KUKA KRL program: EPS_2_25716_MHDR03_A_20250926070354.src

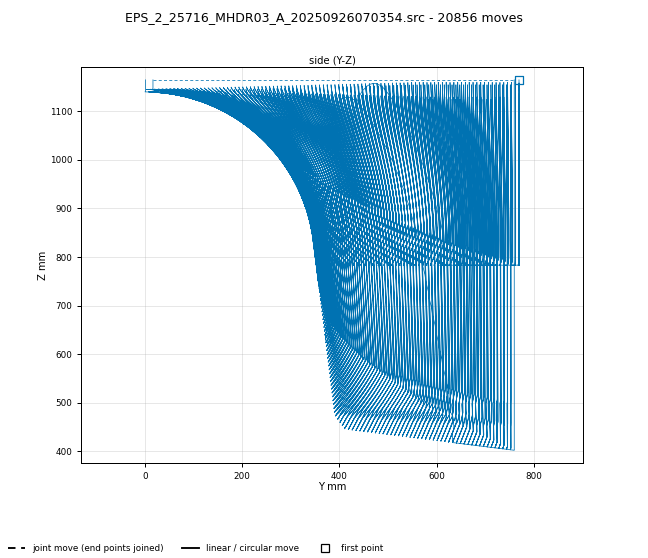
[picture p0: tool path of EPS_2_25716_MHDR03_A_20250926070354.src, 20856 of 20858 moves have a stored position in this frame; points joined in program order, loops and branches not executed]
&ACCESS RVP
&REL 4
&COMMENT QRS 19112012
&PARAM EDITMASK = *
DEF PART()
EXT BAS (BAS_COMMAND :IN,REAL :IN )
INT I
BAS (#INITMOV,0 )

;KUKA QRS Post kuka4.cps  Date:22-06-2017 !

File_ID=2852

QRS_PRE_INIT()

;Init var - Until changes are made in qrs_pre_init
Outlet_Square_prg=0
Inlet_1_Square_prg=0
Inlet_2_Square_prg=0
Inlet_3_Square_prg=0
Inlet_4_Square_prg=0
Inlet_5_Square_prg=0

Outlet_1={X 0.000, Y 562.000, Z 811.500, B 0.000, E1 0.000 }
Inlet_1={X 0.000, Y 582.000, Z 819.500, B 0.000, E1 180.000 }
Outlet_1_type=686
Inlet_1_type=610
;QRS#1=Sidecore dimensions
;QRS#2=675-27" Concrete
;QRS#3=600-24" Concrete
;QRS#4=
;QRS#5=
;QRS#6=
;QRS#7=
;QRS#8=
;QRS#9=S306-38L
;QRS#10=S306-34L
;QRS#11=
;QRS#12=
;QRS#13=
;QRS#14=
;QRS#15=
;QRS#16=1524x152x1600 5,25'
;QRS#17=EPS Height
;QRS#18=1154,5
;QRS#19=*
;QRS#20= UPDATED VERSION 22-06-2017
;QRS#21=*
Outlet_Square=0550
Inlet_1_Square=0450
Inlet_2_Square=0
Inlet_3_Square=0
Inlet_4_Square=0
Inlet_5_Square=0
Mill_Square=1
Outlet_Square_Prg=265
Inlet_1_Square_prg=264

QRS_INIT()

$ADVANCE=5

; T1
PTP {E1 171.915,E2 171.915}
PTP {X 0,Y 769.686,A -85,B 0,C 180,E1 171.915,E2 171.915,E3 0,E4 0,E5 0,E6 0}
QRS_SPEED_INIT()
LIN {X 0,Y 769.686,Z 1164.5,A -85,B 0,C 180,E1 171.915,E2 171.915,E3 0,E4 0,E5 0,E6 0} C_VEL
LIN {X 0,Y 769.686,Z 785.31,A -85,B 0,C 180,E1 171.915,E2 171.915} C_VEL
LIN {X 0,Y 769.694,Z 783.31,A -85,B 0,C 180,E1 172.064,E2 172.064} C_VEL
LIN {X 0,Y 770.026,Z 783.31,A -85,B 0,C 180,E1 173.477,E2 173.477} C_VEL
LIN {X 0,Y 770.008,Z 783.31,A -85,B 0,C 180,E1 177.209,E2 177.209} C_VEL
LIN {X 0,Y 770.018,Z 783.31,A -85,B 0,C 180,E1 180.93,E2 180.93} C_VEL
LIN {X 0,Y 769.994,Z 783.31,A -85,B 0,C 180,E1 184.655,E2 184.655} C_VEL
LIN {X 0,Y 770.012,Z 783.31,A -85,B 0,C 180,E1 188.399,E2 188.399} C_VEL
LIN {X 0,Y 770.006,Z 783.31,A -85,B 0,C 180,E1 192.18,E2 192.18} C_VEL
LIN {X 0,Y 769.997,Z 783.31,A -85,B 0,C 180,E1 196.016,E2 196.016} C_VEL
LIN {X 0,Y 769.871,Z 783.31,A -85,B 0,C 180,E1 196.719,E2 196.719} C_VEL
LIN {X 0,Y 769.991,Z 783.31,A -85,B 0,C 180,E1 199.928,E2 199.928} C_VEL
LIN {X 0,Y 769.967,Z 783.31,A -85,B 0,C 180,E1 203.939,E2 203.939} C_VEL
LIN {X 0,Y 769.591,Z 783.31,A -85,B 0,C 180,E1 206.732,E2 206.732} C_VEL
LIN {X 0,Y 769.94,Z 783.31,A -85,B 0,C 180,E1 208.08,E2 208.08} C_VEL
LIN {X 0,Y 769.516,Z 783.31,A -85,B 0,C 180,E1 210.601,E2 210.601} C_VEL
LIN {X 0,Y 769.912,Z 783.31,A -85,B 0,C 180,E1 212.388,E2 212.388} C_VEL
LIN {X 0,Y 769.473,Z 783.31,A -85,B 0,C 180,E1 214.641,E2 214.641} C_VEL
LIN {X 0,Y 770.033,Z 783.31,A -85,B 0,C 180,E1 217.323,E2 217.323} C_VEL
LIN {X 0,Y 769.708,Z 783.31,A -85,B 0,C 180,E1 221.735,E2 221.735} C_VEL
LIN {X 0,Y 769.752,Z 783.31,A -85,B 0,C 180,E1 223.065,E2 223.065} C_VEL
LIN {X 0,Y 769.737,Z 783.31,A -85,B 0,C 180,E1 226.937,E2 226.937} C_VEL
LIN {X 0,Y 769.694,Z 783.31,A -85,B 0,C 180,E1 228.264,E2 228.264} C_VEL
LIN {X 0,Y 770.056,Z 783.31,A -85,B 0,C 180,E1 232.675,E2 232.675} C_VEL
LIN {X 0,Y 769.726,Z 783.31,A -85,B 0,C 180,E1 235.896,E2 235.896} C_VEL
LIN {X 0,Y 769.776,Z 783.31,A -85,B 0,C 180,E1 237.606,E2 237.606} C_VEL
LIN {X 0,Y 770.022,Z 783.31,A -85,B 0,C 180,E1 240.257,E2 240.257} C_VEL
LIN {X 0,Y 769.768,Z 783.31,A -85,B 0,C 180,E1 240.477,E2 240.477} C_VEL
LIN {X 0,Y 767.999,Z 783.31,A -85,B 0,C 180,E1 240.652,E2 240.652} C_VEL
LIN {X 0,Y 768.022,Z 783.933,A -85,B 0,C 180,E1 240.678,E2 240.678} C_VEL
LIN {X 0,Y 769.268,Z 788.284,A -85,B 0,C 180,E1 240.775,E2 240.775} C_VEL
LIN {X 0,Y 769.55,Z 789.73,A -85,B 0,C 180,E1 240.802,E2 240.802} C_VEL
LIN {X 0,Y 769.707,Z 828.612,A -85,B 0,C 180,E1 241.215,E2 241.215} C_VEL
LIN {X 0,Y 769.834,Z 848.893,A -85,B 0,C 180,E1 241.465,E2 241.465} C_VEL
LIN {X 0,Y 769.636,Z 866.973,A -85,B 0,C 180,E1 241.758,E2 241.758} C_VEL
LIN {X 0,Y 769.793,Z 884.542,A -85,B 0,C 180,E1 242.131,E2 242.131} C_VEL
LIN {X 0,Y 769.673,Z 901.057,A -85,B 0,C 180,E1 242.539,E2 242.539} C_VEL
LIN {X 0,Y 769.87,Z 917.184,A -85,B 0,C 180,E1 243.017,E2 243.017} C_VEL
LIN {X 0,Y 769.856,Z 933.115,A -85,B 0,C 180,E1 243.548,E2 243.548} C_VEL
LIN {X 0,Y 769.816,Z 943.907,A -85,B 0,C 180,E1 243.947,E2 243.947} C_VEL
LIN {X 0,Y 769.91,Z 958.612,A -85,B 0,C 180,E1 244.549,E2 244.549} C_VEL
LIN {X 0,Y 769.91,Z 966.436,A -85,B 0,C 180,E1 244.896,E2 244.896} C_VEL
LIN {X 0,Y 769.862,Z 978.838,A -85,B 0,C 180,E1 245.477,E2 245.477} C_VEL
LIN {X 0,Y 769.916,Z 992.577,A -85,B 0,C 180,E1 246.186,E2 246.186} C_VEL
LIN {X 0,Y 769.931,Z 1006.072,A -85,B 0,C 180,E1 246.947,E2 246.947} C_VEL
LIN {X 0,Y 769.916,Z 1018.978,A -85,B 0,C 180,E1 247.739,E2 247.739} C_VEL
LIN {X 0,Y 769.895,Z 1031.838,A -85,B 0,C 180,E1 248.599,E2 248.599} C_VEL
LIN {X 0,Y 769.943,Z 1043.698,A -85,B 0,C 180,E1 249.463,E2 249.463} C_VEL
LIN {X 0,Y 769.918,Z 1056.014,A -85,B 0,C 180,E1 250.441,E2 250.441} C_VEL
LIN {X 0,Y 769.89,Z 1066.051,A -85,B 0,C 180,E1 251.302,E2 251.302} C_VEL
LIN {X 0,Y 769.98,Z 1077.133,A -85,B 0,C 180,E1 252.343,E2 252.343} C_VEL
LIN {X 0,Y 769.834,Z 1086.51,A -85,B 0,C 180,E1 253.29,E2 253.29} C_VEL
LIN {X 0,Y 769.849,Z 1096.259,A -85,B 0,C 180,E1 254.375,E2 254.375} C_VEL
LIN {X 0,Y 769.966,Z 1105.17,A -85,B 0,C 180,E1 255.468,E2 255.468} C_VEL
LIN {X 0,Y 769.773,Z 1113.783,A -85,B 0,C 180,E1 256.624,E2 256.624} C_VEL
LIN {X 0,Y 769.792,Z 1120.236,A -85,B 0,C 180,E1 257.578,E2 257.578} C_VEL
LIN {X 0,Y 769.971,Z 1127.408,A -85,B 0,C 180,E1 258.769,E2 258.769} C_VEL
LIN {X 0,Y 769.802,Z 1133.795,A -85,B 0,C 180,E1 259.949,E2 259.949} C_VEL
LIN {X 0,Y 769.935,Z 1140.321,A -85,B 0,C 180,E1 261.365,E2 261.365} C_VEL
LIN {X 0,Y 769.915,Z 1143.557,A -85,B 0,C 180,E1 262.172,E2 262.172} C_VEL
LIN {X 0,Y 769.781,Z 1146.098,A -85,B 0,C 180,E1 262.858,E2 262.858} C_VEL
LIN {X 0,Y 769.778,Z 1149.359,A -85,B 0,C 180,E1 263.849,E2 263.849} C_VEL
LIN {X 0,Y 769.874,Z 1151.367,A -85,B 0,C 180,E1 264.598,E2 264.598} C_VEL
LIN {X 0,Y 769.914,Z 1153.173,A -85,B 0,C 180,E1 265.345,E2 265.345} C_VEL
LIN {X 0,Y 769.718,Z 1155.452,A -85,B 0,C 180,E1 266.463,E2 266.463} C_VEL
LIN {X 0,Y 769.72,Z 1156.563,A -85,B 0,C 180,E1 267.208,E2 267.208} C_VEL
LIN {X 0,Y 769.828,Z 1157.375,A -85,B 0,C 180,E1 267.953,E2 267.953} C_VEL
LIN {X 0,Y 769.875,Z 1158.173,A -85,B 0,C 180,E1 269.07,E2 269.07} C_VEL
LIN {X 0,Y 769.75,Z 1158.207,A -85,B 0,C 180,E1 270.93,E2 270.93} C_VEL
LIN {X 0,Y 769.983,Z 1157.332,A -85,B 0,C 180,E1 272.046,E2 272.046} C_VEL
LIN {X 0,Y 769.854,Z 1156.527,A -85,B 0,C 180,E1 272.791,E2 272.791} C_VEL
LIN {X 0,Y 769.764,Z 1155.44,A -85,B 0,C 180,E1 273.537,E2 273.537} C_VEL
LIN {X 0,Y 769.915,Z 1152.382,A -85,B 0,C 180,E1 275.029,E2 275.029} C_VEL
LIN {X 0,Y 769.886,Z 1150.344,A -85,B 0,C 180,E1 275.776,E2 275.776} C_VEL
LIN {X 0,Y 769.765,Z 1148.176,A -85,B 0,C 180,E1 276.525,E2 276.525} C_VEL
LIN {X 0,Y 769.743,Z 1145.274,A -85,B 0,C 180,E1 277.392,E2 277.392} C_VEL
LIN {X 0,Y 769.948,Z 1139.305,A -85,B 0,C 180,E1 278.87,E2 278.87} C_VEL
LIN {X 0,Y 769.75,Z 1133.807,A -85,B 0,C 180,E1 280.051,E2 280.051} C_VEL
LIN {X 0,Y 769.818,Z 1127.44,A -85,B 0,C 180,E1 281.233,E2 281.233} C_VEL
LIN {X 0,Y 769.954,Z 1121.667,A -85,B 0,C 180,E1 282.181,E2 282.181} C_VEL
LIN {X 0,Y 769.843,Z 1116.993,A -85,B 0,C 180,E1 282.897,E2 282.897} C_VEL
LIN {X 0,Y 769.807,Z 1112.103,A -85,B 0,C 180,E1 283.615,E2 283.615} C_VEL
LIN {X 0,Y 769.951,Z 1102.998,A -85,B 0,C 180,E1 284.806,E2 284.806} C_VEL
LIN {X 0,Y 769.846,Z 1094.002,A -85,B 0,C 180,E1 285.885,E2 285.885} C_VEL
LIN {X 0,Y 769.836,Z 1084.723,A -85,B 0,C 180,E1 286.898,E2 286.898} C_VEL
LIN {X 0,Y 769.967,Z 1073.994,A -85,B 0,C 180,E1 287.962,E2 287.962} C_VEL
LIN {X 0,Y 769.883,Z 1063.259,A -85,B 0,C 180,E1 288.944,E2 288.944} C_VEL
LIN {X 0,Y 769.915,Z 1053.038,A -85,B 0,C 180,E1 289.806,E2 289.806} C_VEL
LIN {X 0,Y 769.961,Z 1041.658,A -85,B 0,C 180,E1 290.69,E2 290.69} C_VEL
LIN {X 0,Y 769.906,Z 1029.266,A -85,B 0,C 180,E1 291.578,E2 291.578} C_VEL
LIN {X 0,Y 769.903,Z 1016.603,A -85,B 0,C 180,E1 292.412,E2 292.412} C_VEL
LIN {X 0,Y 769.92,Z 1002.799,A -85,B 0,C 180,E1 293.243,E2 293.243} C_VEL
LIN {X 0,Y 769.909,Z 988.614,A -85,B 0,C 180,E1 294.024,E2 294.024} C_VEL
LIN {X 0,Y 769.846,Z 975.459,A -85,B 0,C 180,E1 294.69,E2 294.69} C_VEL
LIN {X 0,Y 769.908,Z 960.966,A -85,B 0,C 180,E1 295.353,E2 295.353} C_VEL
LIN {X 0,Y 769.866,Z 944.041,A -85,B 0,C 180,E1 296.047,E2 296.047} C_VEL
LIN {X 0,Y 769.796,Z 931.365,A -85,B 0,C 180,E1 296.519,E2 296.519} C_VEL
LIN {X 0,Y 769.894,Z 913.334,A -85,B 0,C 180,E1 297.102,E2 297.102} C_VEL
LIN {X 0,Y 769.78,Z 896.592,A -85,B 0,C 180,E1 297.576,E2 297.576} C_VEL
LIN {X 0,Y 769.701,Z 887.337,A -85,B 0,C 180,E1 297.804,E2 297.804} C_VEL
LIN {X 0,Y 769.825,Z 878.224,A -85,B 0,C 180,E1 298.006,E2 298.006} C_VEL
LIN {X 0,Y 769.846,Z 863.646,A -85,B 0,C 180,E1 298.294,E2 298.294} C_VEL
LIN {X 0,Y 769.602,Z 846.73,A -85,B 0,C 180,E1 298.572,E2 298.572} C_VEL
LIN {X 0,Y 769.68,Z 827.338,A -85,B 0,C 180,E1 298.799,E2 298.799} C_VEL
LIN {X 0,Y 769.587,Z 792.326,A -85,B 0,C 180,E1 299.169,E2 299.169} C_VEL
LIN {X 0,Y 769.462,Z 789.243,A -85,B 0,C 180,E1 299.206,E2 299.206} C_VEL
LIN {X 0,Y 768.376,Z 784.955,A -85,B 0,C 180,E1 299.297,E2 299.297} C_VEL
LIN {X 0,Y 767.908,Z 783.31,A -85,B 0,C 180,E1 299.343,E2 299.343} C_VEL
LIN {X 0,Y 769.576,Z 783.31,A -85,B 0,C 180,E1 299.487,E2 299.487} C_VEL
LIN {X 0,Y 770.036,Z 783.31,A -85,B 0,C 180,E1 299.696,E2 299.696} C_VEL
LIN {X 0,Y 769.963,Z 783.31,A -85,B 0,C 180,E1 302.386,E2 302.386} C_VEL
LIN {X 0,Y 769.484,Z 783.31,A -85,B 0,C 180,E1 304.641,E2 304.641} C_VEL
LIN {X 0,Y 770.058,Z 783.31,A -85,B 0,C 180,E1 307.325,E2 307.325} C_VEL
LIN {X 0,Y 769.794,Z 783.31,A -85,B 0,C 180,E1 311.729,E2 311.729} C_VEL
LIN {X 0,Y 769.849,Z 783.31,A -85,B 0,C 180,E1 313.072,E2 313.072} C_VEL
LIN {X 0,Y 769.85,Z 783.31,A -85,B 0,C 180,E1 314.269,E2 314.269} C_VEL
LIN {X 0,Y 769.763,Z 783.31,A -85,B 0,C 180,E1 315.725,E2 315.725} C_VEL
LIN {X 0,Y 769.779,Z 783.31,A -85,B 0,C 180,E1 319.732,E2 319.732} C_VEL
LIN {X 0,Y 769.826,Z 783.31,A -85,B 0,C 180,E1 320.72,E2 320.72} C_VEL
LIN {X 0,Y 769.435,Z 783.31,A -85,B 0,C 180,E1 323.062,E2 323.062} C_VEL
LIN {X 0,Y 769.867,Z 783.31,A -85,B 0,C 180,E1 325.379,E2 325.379} C_VEL
LIN {X 0,Y 770.015,Z 783.31,A -85,B 0,C 180,E1 329.336,E2 329.336} C_VEL
LIN {X 0,Y 769.861,Z 783.31,A -85,B 0,C 180,E1 333.228,E2 333.228} C_VEL
LIN {X 0,Y 769.954,Z 783.31,A -85,B 0,C 180,E1 334.009,E2 334.009} C_VEL
LIN {X 0,Y 770.01,Z 783.31,A -85,B 0,C 180,E1 337.683,E2 337.683} C_VEL
LIN {X 0,Y 769.98,Z 783.31,A -85,B 0,C 180,E1 338.081,E2 338.081} C_VEL
LIN {X 0,Y 770,Z 783.31,A -85,B 0,C 180,E1 342.039,E2 342.039} C_VEL
LIN {X 0,Y 769.707,Z 783.31,A -85,B 0,C 180,E1 343.978,E2 343.978} C_VEL
LIN {X 0,Y 769.796,Z 783.31,A -85,B 0,C 180,E1 345.906,E2 345.906} C_VEL
LIN {X 0,Y 770.015,Z 783.31,A -85,B 0,C 180,E1 349.716,E2 349.716} C_VEL
LIN {X 0,Y 769.998,Z 783.31,A -85,B 0,C 180,E1 353.477,E2 353.477} C_VEL
LIN {X 0,Y 770.007,Z 783.31,A -85,B 0,C 180,E1 357.209,E2 357.209} C_VEL
LIN {X 0,Y 769.992,Z 783.31,A -85,B 0,C 180,E1 360.93,E2 360.93} C_VEL
LIN {X 0,Y 770.022,Z 783.31,A -85,B 0,C 180,E1 364.655,E2 364.655} C_VEL
LIN {X 0,Y 770.009,Z 783.31,A -85,B 0,C 180,E1 368.399,E2 368.399} C_VEL
LIN {X 0,Y 770.002,Z 783.31,A -85,B 0,C 180,E1 372.18,E2 372.18} C_VEL
LIN {X 0,Y 769.963,Z 783.31,A -85,B 0,C 180,E1 376.017,E2 376.017} C_VEL
LIN {X 0,Y 769.575,Z 783.31,A -85,B 0,C 180,E1 377.971,E2 377.971} C_VEL
LIN {X 0,Y 769.931,Z 783.31,A -85,B 0,C 180,E1 379.929,E2 379.929} C_VEL
LIN {X 0,Y 769.547,Z 783.31,A -85,B 0,C 180,E1 382.233,E2 382.233} C_VEL
LIN {X 0,Y 769.894,Z 783.31,A -85,B 0,C 180,E1 383.942,E2 383.942} C_VEL
LIN {X 0,Y 769.539,Z 783.31,A -85,B 0,C 180,E1 386.724,E2 386.724} C_VEL
LIN {X 0,Y 769.895,Z 783.31,A -85,B 0,C 180,E1 388.082,E2 388.082} C_VEL
LIN {X 0,Y 769.51,Z 783.31,A -85,B 0,C 180,E1 390.601,E2 390.601} C_VEL
LIN {X 0,Y 769.898,Z 783.31,A -85,B 0,C 180,E1 392.389,E2 392.389} C_VEL
LIN {X 0,Y 769.447,Z 783.31,A -85,B 0,C 180,E1 394.643,E2 394.643} C_VEL
LIN {X 0,Y 769.995,Z 783.31,A -85,B 0,C 180,E1 397.319,E2 397.319} C_VEL
LIN {X 0,Y 769.732,Z 783.31,A -85,B 0,C 180,E1 401.733,E2 401.733} C_VEL
LIN {X 0,Y 769.804,Z 783.31,A -85,B 0,C 180,E1 403.069,E2 403.069} C_VEL
LIN {X 0,Y 769.812,Z 783.31,A -85,B 0,C 180,E1 404.272,E2 404.272} C_VEL
LIN {X 0,Y 769.735,Z 783.31,A -85,B 0,C 180,E1 405.723,E2 405.723} C_VEL
LIN {X 0,Y 769.736,Z 783.31,A -85,B 0,C 180,E1 409.736,E2 409.736} C_VEL
LIN {X 0,Y 769.771,Z 783.31,A -85,B 0,C 180,E1 410.717,E2 410.717} C_VEL
LIN {X 0,Y 769.411,Z 783.31,A -85,B 0,C 180,E1 413.061,E2 413.061} C_VEL
LIN {X 0,Y 769.871,Z 783.31,A -85,B 0,C 180,E1 415.379,E2 415.379} C_VEL
LIN {X 0,Y 770.03,Z 783.31,A -85,B 0,C 180,E1 419.334,E2 419.334} C_VEL
LIN {X 0,Y 769.98,Z 783.31,A -85,B 0,C 180,E1 423.211,E2 423.211} C_VEL
LIN {X 0,Y 769.96,Z 783.31,A -85,B 0,C 180,E1 423.598,E2 423.598} C_VEL
LIN {X 0,Y 769.249,Z 783.341,A -85,B 0,C 180,E1 423.817,E2 423.817} C_VEL
LIN {X 0,Y 769.67,Z 784.885,A -85,B 0,C 180,E1 423.848,E2 423.848} C_VEL
LIN {X 0,Y 769.75,Z 839.545,A -85,B 0,C 180,E1 424.413,E2 424.413} C_VEL
LIN {X 0,Y 769.691,Z 849.688,A -85,B 0,C 180,E1 424.533,E2 424.533} C_VEL
LIN {X 0,Y 769.896,Z 867.739,A -85,B 0,C 180,E1 424.833,E2 424.833} C_VEL
LIN {X 0,Y 769.825,Z 882.042,A -85,B 0,C 180,E1 425.12,E2 425.12} C_VEL
LIN {X 0,Y 769.867,Z 892.592,A -85,B 0,C 180,E1 425.372,E2 425.372} C_VEL
LIN {X 0,Y 769.955,Z 909.72,A -85,B 0,C 180,E1 425.842,E2 425.842} C_VEL
LIN {X 0,Y 769.817,Z 926.241,A -85,B 0,C 180,E1 426.374,E2 426.374} C_VEL
LIN {X 0,Y 769.927,Z 939.997,A -85,B 0,C 180,E1 426.884,E2 426.884} C_VEL
LIN {X 0,Y 769.942,Z 953.271,A -85,B 0,C 180,E1 427.43,E2 427.43} C_VEL
LIN {X 0,Y 769.883,Z 966.329,A -85,B 0,C 180,E1 428.023,E2 428.023} C_VEL
LIN {X 0,Y 769.932,Z 980.498,A -85,B 0,C 180,E1 428.744,E2 428.744} C_VEL
LIN {X 0,Y 769.938,Z 991.631,A -85,B 0,C 180,E1 429.36,E2 429.36} C_VEL
LIN {X 0,Y 769.92,Z 1003.392,A -85,B 0,C 180,E1 430.07,E2 430.07} C_VEL
LIN {X 0,Y 769.899,Z 1014.62,A -85,B 0,C 180,E1 430.81,E2 430.81} C_VEL
LIN {X 0,Y 769.914,Z 1026.499,A -85,B 0,C 180,E1 431.67,E2 431.67} C_VEL
LIN {X 0,Y 769.954,Z 1036.883,A -85,B 0,C 180,E1 432.49,E2 432.49} C_VEL
LIN {X 0,Y 769.878,Z 1046.144,A -85,B 0,C 180,E1 433.28,E2 433.28} C_VEL
LIN {X 0,Y 769.886,Z 1055.305,A -85,B 0,C 180,E1 434.13,E2 434.13} C_VEL
LIN {X 0,Y 769.967,Z 1064.552,A -85,B 0,C 180,E1 435.071,E2 435.071} C_VEL
LIN {X 0,Y 769.829,Z 1073.195,A -85,B 0,C 180,E1 436.026,E2 436.026} C_VEL
LIN {X 0,Y 769.837,Z 1080.137,A -85,B 0,C 180,E1 436.864,E2 436.864} C_VEL
LIN {X 0,Y 769.979,Z 1087.29,A -85,B 0,C 180,E1 437.819,E2 437.819} C_VEL
LIN {X 0,Y 769.823,Z 1095.291,A -85,B 0,C 180,E1 439.004,E2 439.004} C_VEL
LIN {X 0,Y 769.817,Z 1101.007,A -85,B 0,C 180,E1 439.95,E2 439.95} C_VEL
LIN {X 0,Y 769.967,Z 1107.201,A -85,B 0,C 180,E1 441.13,E2 441.13} C_VEL
LIN {X 0,Y 769.776,Z 1112.482,A -85,B 0,C 180,E1 442.273,E2 442.273} C_VEL
LIN {X 0,Y 769.779,Z 1116.16,A -85,B 0,C 180,E1 443.191,E2 443.191} C_VEL
LIN {X 0,Y 769.955,Z 1119.598,A -85,B 0,C 180,E1 444.224,E2 444.224} C_VEL
LIN {X 0,Y 769.795,Z 1122.766,A -85,B 0,C 180,E1 445.344,E2 445.344} C_VEL
LIN {X 0,Y 769.781,Z 1125.197,A -85,B 0,C 180,E1 446.463,E2 446.463} C_VEL
LIN {X 0,Y 769.891,Z 1126.354,A -85,B 0,C 180,E1 447.209,E2 447.209} C_VEL
LIN {X 0,Y 769.92,Z 1127.321,A -85,B 0,C 180,E1 447.954,E2 447.954} C_VEL
LIN {X 0,Y 769.761,Z 1128.221,A -85,B 0,C 180,E1 449.07,E2 449.07} C_VEL
LIN {X 0,Y 769.988,Z 1128.134,A -85,B 0,C 180,E1 450.93,E2 450.93} C_VEL
LIN {X 0,Y 769.867,Z 1127.258,A -85,B 0,C 180,E1 452.047,E2 452.047} C_VEL
LIN {X 0,Y 769.876,Z 1126.224,A -85,B 0,C 180,E1 452.791,E2 452.791} C_VEL
LIN {X 0,Y 769.982,Z 1124.952,A -85,B 0,C 180,E1 453.536,E2 453.536} C_VEL
LIN {X 0,Y 769.773,Z 1122.524,A -85,B 0,C 180,E1 454.656,E2 454.656} C_VEL
LIN {X 0,Y 769.789,Z 1119.337,A -85,B 0,C 180,E1 455.777,E2 455.777} C_VEL
LIN {X 0,Y 769.977,Z 1115.754,A -85,B 0,C 180,E1 456.806,E2 456.806} C_VEL
LIN {X 0,Y 769.834,Z 1112.134,A -85,B 0,C 180,E1 457.721,E2 457.721} C_VEL
LIN {X 0,Y 769.821,Z 1106.816,A -85,B 0,C 180,E1 458.872,E2 458.872} C_VEL
LIN {X 0,Y 769.96,Z 1100.444,A -85,B 0,C 180,E1 460.048,E2 460.048} C_VEL
LIN {X 0,Y 769.817,Z 1094.749,A -85,B 0,C 180,E1 460.996,E2 460.996} C_VEL
LIN {X 0,Y 769.85,Z 1086.637,A -85,B 0,C 180,E1 462.183,E2 462.183} C_VEL
LIN {X 0,Y 769.954,Z 1078.394,A -85,B 0,C 180,E1 463.254,E2 463.254} C_VEL
LIN {X 0,Y 769.83,Z 1070.123,A -85,B 0,C 180,E1 464.235,E2 464.235} C_VEL
LIN {X 0,Y 769.861,Z 1062.195,A -85,B 0,C 180,E1 465.093,E2 465.093} C_VEL
LIN {X 0,Y 769.982,Z 1052.807,A -85,B 0,C 180,E1 466.017,E2 466.017} C_VEL
LIN {X 0,Y 769.897,Z 1042.887,A -85,B 0,C 180,E1 466.916,E2 466.916} C_VEL
LIN {X 0,Y 769.891,Z 1033.948,A -85,B 0,C 180,E1 467.664,E2 467.664} C_VEL
LIN {X 0,Y 769.959,Z 1023.69,A -85,B 0,C 180,E1 468.451,E2 468.451} C_VEL
LIN {X 0,Y 769.936,Z 1011.438,A -85,B 0,C 180,E1 469.312,E2 469.312} C_VEL
LIN {X 0,Y 769.918,Z 1000.662,A -85,B 0,C 180,E1 470.009,E2 470.009} C_VEL
LIN {X 0,Y 769.899,Z 988.438,A -85,B 0,C 180,E1 470.732,E2 470.732} C_VEL
LIN {X 0,Y 769.925,Z 975.866,A -85,B 0,C 180,E1 471.409,E2 471.409} C_VEL
LIN {X 0,Y 769.921,Z 963.055,A -85,B 0,C 180,E1 472.039,E2 472.039} C_VEL
LIN {X 0,Y 769.849,Z 949.556,A -85,B 0,C 180,E1 472.641,E2 472.641} C_VEL
LIN {X 0,Y 769.935,Z 935.996,A -85,B 0,C 180,E1 473.179,E2 473.179} C_VEL
LIN {X 0,Y 769.929,Z 921.73,A -85,B 0,C 180,E1 473.686,E2 473.686} C_VEL
LIN {X 0,Y 769.79,Z 908.407,A -85,B 0,C 180,E1 474.111,E2 474.111} C_VEL
LIN {X 0,Y 769.935,Z 893.14,A -85,B 0,C 180,E1 474.523,E2 474.523} C_VEL
LIN {X 0,Y 769.918,Z 878.801,A -85,B 0,C 180,E1 474.858,E2 474.858} C_VEL
LIN {X 0,Y 769.735,Z 864.362,A -85,B 0,C 180,E1 475.145,E2 475.145} C_VEL
LIN {X 0,Y 769.91,Z 847.878,A -85,B 0,C 180,E1 475.391,E2 475.391} C_VEL
LIN {X 0,Y 769.846,Z 830.427,A -85,B 0,C 180,E1 475.593,E2 475.593} C_VEL
LIN {X 0,Y 769.259,Z 783.31,A -85,B 0,C 180,E1 476.094,E2 476.094} C_VEL
LIN {X 0,Y 769.934,Z 783.31,A -85,B 0,C 180,E1 476.198,E2 476.198} C_VEL
LIN {X 0,Y 770.046,Z 783.31,A -85,B 0,C 180,E1 476.399,E2 476.399} C_VEL
LIN {X 0,Y 769.988,Z 783.31,A -85,B 0,C 180,E1 478.078,E2 478.078} C_VEL
LIN {X 0,Y 769.523,Z 783.31,A -85,B 0,C 180,E1 480.602,E2 480.602} C_VEL
LIN {X 0,Y 769.907,Z 783.31,A -85,B 0,C 180,E1 482.388,E2 482.388} C_VEL
LIN {X 0,Y 769.561,Z 783.31,A -85,B 0,C 180,E1 484.086,E2 484.086} C_VEL
LIN {X 0,Y 770.003,Z 783.31,A -85,B 0,C 180,E1 487.32,E2 487.32} C_VEL
LIN {X 0,Y 769.731,Z 783.31,A -85,B 0,C 180,E1 491.733,E2 491.733} C_VEL
LIN {X 0,Y 769.809,Z 783.31,A -85,B 0,C 180,E1 493.069,E2 493.069} C_VEL
LIN {X 0,Y 769.813,Z 783.31,A -85,B 0,C 180,E1 494.271,E2 494.271} C_VEL
LIN {X 0,Y 769.743,Z 783.31,A -85,B 0,C 180,E1 495.723,E2 495.723} C_VEL
LIN {X 0,Y 769.727,Z 783.31,A -85,B 0,C 180,E1 499.736,E2 499.736} C_VEL
LIN {X 0,Y 769.752,Z 783.31,A -85,B 0,C 180,E1 500.715,E2 500.715} C_VEL
LIN {X 0,Y 769.387,Z 783.31,A -85,B 0,C 180,E1 503.059,E2 503.059} C_VEL
LIN {X 0,Y 769.85,Z 783.31,A -85,B 0,C 180,E1 505.378,E2 505.378} C_VEL
LIN {X 0,Y 769.987,Z 783.31,A -85,B 0,C 180,E1 509.339,E2 509.339} C_VEL
LIN {X 0,Y 769.816,Z 783.31,A -85,B 0,C 180,E1 513.235,E2 513.235} C_VEL
LIN {X 0,Y 769.906,Z 783.31,A -85,B 0,C 180,E1 514.007,E2 514.007} C_VEL
LIN {X 0,Y 769.968,Z 783.31,A -85,B 0,C 180,E1 517.691,E2 517.691} C_VEL
LIN {X 0,Y 769.921,Z 783.31,A -85,B 0,C 180,E1 518.079,E2 518.079} C_VEL
LIN {X 0,Y 769.973,Z 783.31,A -85,B 0,C 180,E1 522.038,E2 522.038} C_VEL
LIN {X 0,Y 769.719,Z 783.31,A -85,B 0,C 180,E1 523.978,E2 523.978} C_VEL
LIN {X 0,Y 769.82,Z 783.31,A -85,B 0,C 180,E1 525.906,E2 525.906} C_VEL
LIN {X 0,Y 770.045,Z 783.31,A -85,B 0,C 180,E1 529.716,E2 529.716} C_VEL
LIN {X 0,Y 769.694,Z 783.31,A -85,B 0,C 180,E1 532.064,E2 532.064} C_VEL
LIN {X 0,Y 765.83,Z 783.31,A -85,B 0,C 180,E1 533.34,E2 533.34} C_VEL
LIN {X 0,Y 761.787,Z 783.31,A -85,B 0,C 180,E1 534.629,E2 534.629} C_VEL
LIN {X 0,Y 761.742,Z 783.31,A -85,B 0,C 180,E1 538.856,E2 538.856} C_VEL
LIN {X 0,Y 761.741,Z 783.31,A -85,B 0,C 180,E1 542.275,E2 542.275} C_VEL
LIN {X 0,Y 761.746,Z 783.31,A -85,B 0,C 180,E1 545.986,E2 545.986} C_VEL
LIN {X 0,Y 761.697,Z 783.31,A -85,B 0,C 180,E1 550.308,E2 550.308} C_VEL
LIN {X 0,Y 761.695,Z 783.31,A -85,B 0,C 180,E1 553.804,E2 553.804} C_VEL
LIN {X 0,Y 761.804,Z 783.31,A -85,B 0,C 180,E1 557.352,E2 557.352} C_VEL
LIN {X 0,Y 761.737,Z 783.31,A -85,B 0,C 180,E1 560.973,E2 560.973} C_VEL
LIN {X 0,Y 761.793,Z 783.31,A -85,B 0,C 180,E1 564.681,E2 564.681} C_VEL
LIN {X 0,Y 761.743,Z 783.31,A -85,B 0,C 180,E1 568.93,E2 568.93} C_VEL
LIN {X 0,Y 761.709,Z 783.31,A -85,B 0,C 180,E1 573.336,E2 573.336} C_VEL
LIN {X 0,Y 761.761,Z 783.31,A -85,B 0,C 180,E1 578.059,E2 578.059} C_VEL
LIN {X 0,Y 761.819,Z 783.31,A -85,B 0,C 180,E1 582.617,E2 582.617} C_VEL
LIN {X 0,Y 761.791,Z 783.31,A -85,B 0,C 180,E1 587.448,E2 587.448} C_VEL
LIN {X 0,Y 761.906,Z 783.31,A -85,B 0,C 180,E1 593.372,E2 593.372} C_VEL
LIN {X 0,Y 761.81,Z 783.31,A -85,B 0,C 180,E1 598.768,E2 598.768} C_VEL
LIN {X 0,Y 761.34,Z 783.31,A -85,B 0,C 180,E1 600.334,E2 600.334} C_VEL
LIN {X 0,Y 762.671,Z 794.401,A -85,B 0,C 180,E1 600.563,E2 600.563} C_VEL
LIN {X 0,Y 762.736,Z 862.317,A -85,B 0,C 180,E1 601.396,E2 601.396} C_VEL
LIN {X 0,Y 762.643,Z 906.034,A -85,B 0,C 180,E1 602.408,E2 602.408} C_VEL
LIN {X 0,Y 762.612,Z 948.961,A -85,B 0,C 180,E1 603.882,E2 603.882} C_VEL
LIN {X 0,Y 762.519,Z 991.458,A -85,B 0,C 180,E1 605.878,E2 605.878} C_VEL
LIN {X 0,Y 762.316,Z 1031.466,A -85,B 0,C 180,E1 608.348,E2 608.348} C_VEL
LIN {X 0,Y 762.188,Z 1066.636,A -85,B 0,C 180,E1 611.152,E2 611.152} C_VEL
LIN {X 0,Y 762.091,Z 1095.886,A -85,B 0,C 180,E1 614.134,E2 614.134} C_VEL
LIN {X 0,Y 761.966,Z 1120.139,A -85,B 0,C 180,E1 617.364,E2 617.364} C_VEL
LIN {X 0,Y 762.006,Z 1136.484,A -85,B 0,C 180,E1 620.269,E2 620.269} C_VEL
LIN {X 0,Y 761.959,Z 1149.189,A -85,B 0,C 180,E1 623.454,E2 623.454} C_VEL
LIN {X 0,Y 761.907,Z 1156.65,A -85,B 0,C 180,E1 626.579,E2 626.579} C_VEL
LIN {X 0,Y 761.941,Z 1159.5,A -85,B 0,C 180,E1 629.999,E2 629.999} C_VEL
LIN {X 0,Y 761.964,Z 1156.652,A -85,B 0,C 180,E1 633.419,E2 633.419} C_VEL
LIN {X 0,Y 762.008,Z 1150.104,A -85,B 0,C 180,E1 636.267,E2 636.267} C_VEL
LIN {X 0,Y 761.986,Z 1136.494,A -85,B 0,C 180,E1 639.73,E2 639.73} C_VEL
LIN {X 0,Y 762.053,Z 1118.033,A -85,B 0,C 180,E1 642.947,E2 642.947} C_VEL
LIN {X 0,Y 762.078,Z 1094.582,A -85,B 0,C 180,E1 646.012,E2 646.012} C_VEL
LIN {X 0,Y 762.211,Z 1065.026,A -85,B 0,C 180,E1 648.995,E2 648.995} C_VEL
LIN {X 0,Y 762.343,Z 1030.425,A -85,B 0,C 180,E1 651.725,E2 651.725} C_VEL
LIN {X 0,Y 762.512,Z 990.308,A -85,B 0,C 180,E1 654.185,E2 654.185} C_VEL
LIN {X 0,Y 762.649,Z 947.471,A -85,B 0,C 180,E1 656.179,E2 656.179} C_VEL
LIN {X 0,Y 762.742,Z 904.721,A -85,B 0,C 180,E1 657.626,E2 657.626} C_VEL
LIN {X 0,Y 762.846,Z 862.737,A -85,B 0,C 180,E1 658.592,E2 658.592} C_VEL
LIN {X 0,Y 762.707,Z 806.91,A -85,B 0,C 180,E1 659.303,E2 659.303} C_VEL
LIN {X 0,Y 761.982,Z 788.522,A -85,B 0,C 180,E1 659.529,E2 659.529} C_VEL
LIN {X 0,Y 761.156,Z 783.31,A -85,B 0,C 180,E1 659.65,E2 659.65} C_VEL
LIN {X 0,Y 762.115,Z 783.31,A -85,B 0,C 180,E1 659.802,E2 659.802} C_VEL
LIN {X 0,Y 761.637,Z 783.31,A -85,B 0,C 180,E1 663.849,E2 663.849} C_VEL
LIN {X 0,Y 761.824,Z 783.31,A -85,B 0,C 180,E1 668.063,E2 668.063} C_VEL
LIN {X 0,Y 761.908,Z 783.31,A -85,B 0,C 180,E1 672.637,E2 672.637} C_VEL
LIN {X 0,Y 761.794,Z 783.31,A -85,B 0,C 180,E1 675.894,E2 675.894} C_VEL
LIN {X 0,Y 761.871,Z 783.31,A -85,B 0,C 180,E1 680.859,E2 680.859} C_VEL
LIN {X 0,Y 761.704,Z 783.31,A -85,B 0,C 180,E1 686.162,E2 686.162} C_VEL
LIN {X 0,Y 761.789,Z 783.31,A -85,B 0,C 180,E1 690.191,E2 690.191} C_VEL
LIN {X 0,Y 762.027,Z 783.31,A -85,B 0,C 180,E1 694.067,E2 694.067} C_VEL
LIN {X 0,Y 762.125,Z 783.31,A -85,B 0,C 180,E1 697.813,E2 697.813} C_VEL
LIN {X 0,Y 761.926,Z 783.31,A -85,B 0,C 180,E1 702.651,E2 702.651} C_VEL
LIN {X 0,Y 761.608,Z 783.31,A -85,B 0,C 180,E1 707.365,E2 707.365} C_VEL
LIN {X 0,Y 761.765,Z 783.31,A -85,B 0,C 180,E1 710.849,E2 710.849} C_VEL
LIN {X 0,Y 761.819,Z 783.31,A -85,B 0,C 180,E1 714.298,E2 714.298} C_VEL
LIN {X 0,Y 761.702,Z 783.31,A -85,B 0,C 180,E1 718.865,E2 718.865} C_VEL
LIN {X 0,Y 761.738,Z 783.31,A -85,B 0,C 180,E1 722.284,E2 722.284} C_VEL
LIN {X 0,Y 761.756,Z 783.31,A -85,B 0,C 180,E1 726.011,E2 726.011} C_VEL
LIN {X 0,Y 761.71,Z 783.31,A -85,B 0,C 180,E1 730.316,E2 730.316} C_VEL
LIN {X 0,Y 761.67,Z 783.31,A -85,B 0,C 180,E1 733.814,E2 733.814} C_VEL
LIN {X 0,Y 761.704,Z 783.31,A -85,B 0,C 180,E1 737.363,E2 737.363} C_VEL
LIN {X 0,Y 761.701,Z 783.31,A -85,B 0,C 180,E1 740.983,E2 740.983} C_VEL
LIN {X 0,Y 761.727,Z 783.31,A -85,B 0,C 180,E1 744.693,E2 744.693} C_VEL
LIN {X 0,Y 761.722,Z 783.31,A -85,B 0,C 180,E1 748.932,E2 748.932} C_VEL
LIN {X 0,Y 761.667,Z 783.31,A -85,B 0,C 180,E1 753.335,E2 753.335} C_VEL
LIN {X 0,Y 761.734,Z 783.31,A -85,B 0,C 180,E1 758.071,E2 758.071} C_VEL
LIN {X 0,Y 761.834,Z 783.31,A -85,B 0,C 180,E1 762.621,E2 762.621} C_VEL
LIN {X 0,Y 761.772,Z 783.31,A -85,B 0,C 180,E1 765.883,E2 765.883} C_VEL
LIN {X 0,Y 761.823,Z 783.31,A -85,B 0,C 180,E1 770.865,E2 770.865} C_VEL
LIN {X 0,Y 761.712,Z 783.31,A -85,B 0,C 180,E1 776.155,E2 776.155} C_VEL
LIN {X 0,Y 761.83,Z 783.31,A -85,B 0,C 180,E1 780.186,E2 780.186} C_VEL
LIN {X 0,Y 762,Z 783.497,A -85,B 0,C 180,E1 783.55,E2 783.55} C_VEL
LIN {X 0,Y 762.696,Z 862.149,A -85,B 0,C 180,E1 784.48,E2 784.48} C_VEL
LIN {X 0,Y 762.688,Z 902.947,A -85,B 0,C 180,E1 785.406,E2 785.406} C_VEL
LIN {X 0,Y 762.539,Z 940.389,A -85,B 0,C 180,E1 786.663,E2 786.663} C_VEL
LIN {X 0,Y 762.431,Z 978.798,A -85,B 0,C 180,E1 788.431,E2 788.431} C_VEL
LIN {X 0,Y 762.254,Z 1014.897,A -85,B 0,C 180,E1 790.629,E2 790.629} C_VEL
LIN {X 0,Y 762.181,Z 1046.217,A -85,B 0,C 180,E1 793.099,E2 793.099} C_VEL
LIN {X 0,Y 762.081,Z 1073.73,A -85,B 0,C 180,E1 795.905,E2 795.905} C_VEL
LIN {X 0,Y 762.025,Z 1095.461,A -85,B 0,C 180,E1 798.823,E2 798.823} C_VEL
LIN {X 0,Y 761.979,Z 1112.455,A -85,B 0,C 180,E1 802,E2 802} C_VEL
LIN {X 0,Y 762.022,Z 1122.532,A -85,B 0,C 180,E1 804.868,E2 804.868} C_VEL
LIN {X 0,Y 762.083,Z 1128.181,A -85,B 0,C 180,E1 807.722,E2 807.722} C_VEL
LIN {X 0,Y 762.127,Z 1129.116,A -85,B 0,C 180,E1 811.14,E2 811.14} C_VEL
LIN {X 0,Y 762.069,Z 1125.1,A -85,B 0,C 180,E1 813.991,E2 813.991} C_VEL
LIN {X 0,Y 762.096,Z 1115.579,A -85,B 0,C 180,E1 817.139,E2 817.139} C_VEL
LIN {X 0,Y 762.107,Z 1100.156,A -85,B 0,C 180,E1 820.308,E2 820.308} C_VEL
LIN {X 0,Y 762.166,Z 1079.387,A -85,B 0,C 180,E1 823.32,E2 823.32} C_VEL
LIN {X 0,Y 762.234,Z 1053.265,A -85,B 0,C 180,E1 826.159,E2 826.159} C_VEL
LIN {X 0,Y 762.298,Z 1021.984,A -85,B 0,C 180,E1 828.77,E2 828.77} C_VEL
LIN {X 0,Y 762.377,Z 988.156,A -85,B 0,C 180,E1 830.962,E2 830.962} C_VEL
LIN {X 0,Y 762.465,Z 949.445,A -85,B 0,C 180,E1 832.877,E2 832.877} C_VEL
LIN {X 0,Y 762.538,Z 907.416,A -85,B 0,C 180,E1 834.384,E2 834.384} C_VEL
LIN {X 0,Y 762.6,Z 863.769,A -85,B 0,C 180,E1 835.407,E2 835.407} C_VEL
LIN {X 0,Y 762.211,Z 788.184,A -85,B 0,C 180,E1 836.303,E2 836.303} C_VEL
LIN {X 0,Y 762.142,Z 783.31,A -85,B 0,C 180,E1 836.373,E2 836.373} C_VEL
LIN {X 0,Y 761.994,Z 783.31,A -85,B 0,C 180,E1 842.472,E2 842.472} C_VEL
LIN {X 0,Y 761.742,Z 783.31,A -85,B 0,C 180,E1 848.07,E2 848.07} C_VEL
LIN {X 0,Y 761.865,Z 783.31,A -85,B 0,C 180,E1 852.621,E2 852.621} C_VEL
LIN {X 0,Y 761.773,Z 783.31,A -85,B 0,C 180,E1 855.88,E2 855.88} C_VEL
LIN {X 0,Y 761.806,Z 783.31,A -85,B 0,C 180,E1 860.868,E2 860.868} C_VEL
LIN {X 0,Y 761.716,Z 783.31,A -85,B 0,C 180,E1 866.153,E2 866.153} C_VEL
LIN {X 0,Y 761.763,Z 783.31,A -85,B 0,C 180,E1 870.18,E2 870.18} C_VEL
LIN {X 0,Y 762.002,Z 783.31,A -85,B 0,C 180,E1 874.057,E2 874.057} C_VEL
LIN {X 0,Y 762.059,Z 783.31,A -85,B 0,C 180,E1 877.802,E2 877.802} C_VEL
LIN {X 0,Y 761.894,Z 783.31,A -85,B 0,C 180,E1 882.665,E2 882.665} C_VEL
LIN {X 0,Y 761.617,Z 783.31,A -85,B 0,C 180,E1 887.356,E2 887.356} C_VEL
LIN {X 0,Y 761.828,Z 783.31,A -85,B 0,C 180,E1 890.841,E2 890.841} C_VEL
LIN {X 0,Y 761.787,Z 783.31,A -85,B 0,C 180,E1 894.629,E2 894.629} C_VEL
LIN {X 0,Y 757.809,Z 783.31,A -85,B 0,C 180,E1 895.911,E2 895.911} C_VEL
LIN {X 0,Y 753.971,Z 783.31,A -85,B 0,C 180,E1 897.208,E2 897.208} C_VEL
LIN {X 0,Y 753.846,Z 783.31,A -85,B 0,C 180,E1 902.299,E2 902.299} C_VEL
LIN {X 0,Y 753.893,Z 783.31,A -85,B 0,C 180,E1 905.762,E2 905.762} C_VEL
LIN {X 0,Y 753.825,Z 783.31,A -85,B 0,C 180,E1 909.97,E2 909.97} C_VEL
LIN {X 0,Y 753.789,Z 783.31,A -85,B 0,C 180,E1 913.952,E2 913.952} C_VEL
LIN {X 0,Y 753.874,Z 783.31,A -85,B 0,C 180,E1 917.54,E2 917.54} C_VEL
LIN {X 0,Y 753.792,Z 783.31,A -85,B 0,C 180,E1 921.205,E2 921.205} C_VEL
LIN {X 0,Y 753.798,Z 783.31,A -85,B 0,C 180,E1 925.239,E2 925.239} C_VEL
LIN {X 0,Y 753.882,Z 783.31,A -85,B 0,C 180,E1 928.832,E2 928.832} C_VEL
LIN {X 0,Y 753.95,Z 783.31,A -85,B 0,C 180,E1 932.852,E2 932.852} C_VEL
LIN {X 0,Y 754.102,Z 783.31,A -85,B 0,C 180,E1 937.059,E2 937.059} C_VEL
LIN {X 0,Y 753.768,Z 783.31,A -85,B 0,C 180,E1 943.102,E2 943.102} C_VEL
LIN {X 0,Y 753.681,Z 783.31,A -85,B 0,C 180,E1 948.438,E2 948.438} C_VEL
LIN {X 0,Y 753.972,Z 783.31,A -85,B 0,C 180,E1 953.483,E2 953.483} C_VEL
LIN {X 0,Y 753.902,Z 783.31,A -85,B 0,C 180,E1 958.496,E2 958.496} C_VEL
LIN {X 0,Y 754.189,Z 783.31,A -85,B 0,C 180,E1 960.068,E2 960.068} C_VEL
LIN {X 0,Y 755.811,Z 800.454,A -85,B 0,C 180,E1 960.334,E2 960.334} C_VEL
LIN {X 0,Y 755.776,Z 864.219,A -85,B 0,C 180,E1 961.14,E2 961.14} C_VEL
LIN {X 0,Y 755.561,Z 908.581,A -85,B 0,C 180,E1 962.201,E2 962.201} C_VEL
LIN {X 0,Y 755.365,Z 950.451,A -85,B 0,C 180,E1 963.676,E2 963.676} C_VEL
LIN {X 0,Y 755.099,Z 991.457,A -85,B 0,C 180,E1 965.625,E2 965.625} C_VEL
LIN {X 0,Y 754.775,Z 1031.464,A -85,B 0,C 180,E1 968.121,E2 968.121} C_VEL
LIN {X 0,Y 754.526,Z 1064.778,A -85,B 0,C 180,E1 970.782,E2 970.782} C_VEL
LIN {X 0,Y 754.308,Z 1094.368,A -85,B 0,C 180,E1 973.794,E2 973.794} C_VEL
LIN {X 0,Y 754.118,Z 1117.417,A -85,B 0,C 180,E1 976.822,E2 976.822} C_VEL
LIN {X 0,Y 754.129,Z 1135.546,A -85,B 0,C 180,E1 979.962,E2 979.962} C_VEL
LIN {X 0,Y 754.051,Z 1148.156,A -85,B 0,C 180,E1 983.074,E2 983.074} C_VEL
LIN {X 0,Y 754.09,Z 1155.659,A -85,B 0,C 180,E1 985.966,E2 985.966} C_VEL
LIN {X 0,Y 754.133,Z 1159.171,A -85,B 0,C 180,E1 988.848,E2 988.848} C_VEL
LIN {X 0,Y 754.224,Z 1158.221,A -85,B 0,C 180,E1 992.302,E2 992.302} C_VEL
LIN {X 0,Y 754.182,Z 1151.637,A -85,B 0,C 180,E1 995.764,E2 995.764} C_VEL
LIN {X 0,Y 754.21,Z 1140.529,A -85,B 0,C 180,E1 998.956,E2 998.956} C_VEL
LIN {X 0,Y 754.256,Z 1122.036,A -85,B 0,C 180,E1 1002.47,E2 1002.47} C_VEL
LIN {X 0,Y 754.276,Z 1098.013,A -85,B 0,C 180,E1 1005.774,E2 1005.774} C_VEL
LIN {X 0,Y 754.506,Z 1069.881,A -85,B 0,C 180,E1 1008.741,E2 1008.741} C_VEL
LIN {X 0,Y 754.747,Z 1037.775,A -85,B 0,C 180,E1 1011.414,E2 1011.414} C_VEL
LIN {X 0,Y 755.035,Z 1002.305,A -85,B 0,C 180,E1 1013.758,E2 1013.758} C_VEL
LIN {X 0,Y 755.336,Z 962.011,A -85,B 0,C 180,E1 1015.832,E2 1015.832} C_VEL
LIN {X 0,Y 755.639,Z 919.332,A -85,B 0,C 180,E1 1017.462,E2 1017.462} C_VEL
LIN {X 0,Y 755.834,Z 878.464,A -85,B 0,C 180,E1 1018.567,E2 1018.567} C_VEL
LIN {X 0,Y 755.851,Z 835.002,A -85,B 0,C 180,E1 1019.29,E2 1019.29} C_VEL
LIN {X 0,Y 755.023,Z 789.962,A -85,B 0,C 180,E1 1019.813,E2 1019.813} C_VEL
LIN {X 0,Y 754.165,Z 783.31,A -85,B 0,C 180,E1 1019.974,E2 1019.974} C_VEL
LIN {X 0,Y 753.673,Z 783.31,A -85,B 0,C 180,E1 1024.256,E2 1024.256} C_VEL
LIN {X 0,Y 753.826,Z 783.31,A -85,B 0,C 180,E1 1028.396,E2 1028.396} C_VEL
LIN {X 0,Y 754.02,Z 783.31,A -85,B 0,C 180,E1 1033.676,E2 1033.676} C_VEL
LIN {X 0,Y 753.575,Z 783.31,A -85,B 0,C 180,E1 1038.442,E2 1038.442} C_VEL
LIN {X 0,Y 753.625,Z 783.31,A -85,B 0,C 180,E1 1042.914,E2 1042.914} C_VEL
LIN {X 0,Y 753.712,Z 783.31,A -85,B 0,C 180,E1 1047.596,E2 1047.596} C_VEL
LIN {X 0,Y 753.755,Z 783.31,A -85,B 0,C 180,E1 1052.184,E2 1052.184} C_VEL
LIN {X 0,Y 753.858,Z 783.31,A -85,B 0,C 180,E1 1055.042,E2 1055.042} C_VEL
LIN {X 0,Y 753.895,Z 783.31,A -85,B 0,C 180,E1 1058.798,E2 1058.798} C_VEL
LIN {X 0,Y 753.911,Z 783.31,A -85,B 0,C 180,E1 1063.664,E2 1063.664} C_VEL
LIN {X 0,Y 753.761,Z 783.31,A -85,B 0,C 180,E1 1068.409,E2 1068.409} C_VEL
LIN {X 0,Y 753.809,Z 783.31,A -85,B 0,C 180,E1 1071.917,E2 1071.917} C_VEL
LIN {X 0,Y 753.996,Z 783.31,A -85,B 0,C 180,E1 1076.548,E2 1076.548} C_VEL
LIN {X 0,Y 754.099,Z 783.31,A -85,B 0,C 180,E1 1081.155,E2 1081.155} C_VEL
LIN {X 0,Y 753.893,Z 783.31,A -85,B 0,C 180,E1 1085.771,E2 1085.771} C_VEL
LIN {X 0,Y 753.824,Z 783.31,A -85,B 0,C 180,E1 1090.425,E2 1090.425} C_VEL
LIN {X 0,Y 753.862,Z 783.31,A -85,B 0,C 180,E1 1095.149,E2 1095.149} C_VEL
LIN {X 0,Y 754.006,Z 783.31,A -85,B 0,C 180,E1 1099.978,E2 1099.978} C_VEL
LIN {X 0,Y 753.759,Z 783.31,A -85,B 0,C 180,E1 1104.971,E2 1104.971} C_VEL
LIN {X 0,Y 753.839,Z 783.31,A -85,B 0,C 180,E1 1108.843,E2 1108.843} C_VEL
LIN {X 0,Y 753.933,Z 783.31,A -85,B 0,C 180,E1 1112.863,E2 1112.863} C_VEL
LIN {X 0,Y 754.073,Z 783.31,A -85,B 0,C 180,E1 1117.071,E2 1117.071} C_VEL
LIN {X 0,Y 753.911,Z 783.31,A -85,B 0,C 180,E1 1123.104,E2 1123.104} C_VEL
LIN {X 0,Y 753.6,Z 783.31,A -85,B 0,C 180,E1 1126.876,E2 1126.876} C_VEL
LIN {X 0,Y 753.724,Z 783.31,A -85,B 0,C 180,E1 1131.628,E2 1131.628} C_VEL
LIN {X 0,Y 753.773,Z 783.31,A -85,B 0,C 180,E1 1135.75,E2 1135.75} C_VEL
LIN {X 0,Y 753.921,Z 783.31,A -85,B 0,C 180,E1 1139.84,E2 1139.84} C_VEL
LIN {X 0,Y 754.131,Z 783.31,A -85,B 0,C 180,E1 1143.241,E2 1143.241} C_VEL
LIN {X 0,Y 755.495,Z 793.242,A -85,B 0,C 180,E1 1143.407,E2 1143.407} C_VEL
LIN {X 0,Y 755.547,Z 862.74,A -85,B 0,C 180,E1 1144.231,E2 1144.231} C_VEL
LIN {X 0,Y 755.432,Z 903.963,A -85,B 0,C 180,E1 1145.183,E2 1145.183} C_VEL
LIN {X 0,Y 755.152,Z 942.103,A -85,B 0,C 180,E1 1146.493,E2 1146.493} C_VEL
LIN {X 0,Y 754.918,Z 980.174,A -85,B 0,C 180,E1 1148.282,E2 1148.282} C_VEL
LIN {X 0,Y 754.598,Z 1016.21,A -85,B 0,C 180,E1 1150.52,E2 1150.52} C_VEL
LIN {X 0,Y 754.417,Z 1048.074,A -85,B 0,C 180,E1 1153.094,E2 1153.094} C_VEL
LIN {X 0,Y 754.247,Z 1073.727,A -85,B 0,C 180,E1 1155.755,E2 1155.755} C_VEL
LIN {X 0,Y 754.165,Z 1095.458,A -85,B 0,C 180,E1 1158.705,E2 1158.705} C_VEL
LIN {X 0,Y 754.098,Z 1112.453,A -85,B 0,C 180,E1 1161.916,E2 1161.916} C_VEL
LIN {X 0,Y 754.152,Z 1122.532,A -85,B 0,C 180,E1 1164.814,E2 1164.814} C_VEL
LIN {X 0,Y 754.178,Z 1128.181,A -85,B 0,C 180,E1 1167.698,E2 1167.698} C_VEL
LIN {X 0,Y 754.225,Z 1129.117,A -85,B 0,C 180,E1 1171.152,E2 1171.152} C_VEL
LIN {X 0,Y 754.174,Z 1125.102,A -85,B 0,C 180,E1 1174.033,E2 1174.033} C_VEL
LIN {X 0,Y 754.198,Z 1115.581,A -85,B 0,C 180,E1 1177.214,E2 1177.214} C_VEL
LIN {X 0,Y 754.267,Z 1101.635,A -85,B 0,C 180,E1 1180.17,E2 1180.17} C_VEL
LIN {X 0,Y 754.333,Z 1080.027,A -85,B 0,C 180,E1 1183.384,E2 1183.384} C_VEL
LIN {X 0,Y 754.459,Z 1053.271,A -85,B 0,C 180,E1 1186.33,E2 1186.33} C_VEL
LIN {X 0,Y 754.635,Z 1022.079,A -85,B 0,C 180,E1 1188.961,E2 1188.961} C_VEL
LIN {X 0,Y 754.825,Z 988.168,A -85,B 0,C 180,E1 1191.182,E2 1191.182} C_VEL
LIN {X 0,Y 755.086,Z 950.806,A -85,B 0,C 180,E1 1193.058,E2 1193.058} C_VEL
LIN {X 0,Y 755.285,Z 908.632,A -85,B 0,C 180,E1 1194.599,E2 1194.599} C_VEL
LIN {X 0,Y 755.48,Z 863.924,A -85,B 0,C 180,E1 1195.662,E2 1195.662} C_VEL
LIN {X 0,Y 755.12,Z 788.066,A -85,B 0,C 180,E1 1196.571,E2 1196.571} C_VEL
LIN {X 0,Y 754.201,Z 783.31,A -85,B 0,C 180,E1 1196.722,E2 1196.722} C_VEL
LIN {X 0,Y 753.982,Z 783.31,A -85,B 0,C 180,E1 1202.86,E2 1202.86} C_VEL
LIN {X 0,Y 754.091,Z 783.31,A -85,B 0,C 180,E1 1207.07,E2 1207.07} C_VEL
LIN {X 0,Y 753.943,Z 783.31,A -85,B 0,C 180,E1 1213.657,E2 1213.657} C_VEL
LIN {X 0,Y 753.548,Z 783.31,A -85,B 0,C 180,E1 1218.429,E2 1218.429} C_VEL
LIN {X 0,Y 753.584,Z 783.31,A -85,B 0,C 180,E1 1222.9,E2 1222.9} C_VEL
LIN {X 0,Y 753.7,Z 783.31,A -85,B 0,C 180,E1 1227.602,E2 1227.602} C_VEL
LIN {X 0,Y 753.727,Z 783.31,A -85,B 0,C 180,E1 1232.192,E2 1232.192} C_VEL
LIN {X 0,Y 753.799,Z 783.31,A -85,B 0,C 180,E1 1236.294,E2 1236.294} C_VEL
LIN {X 0,Y 753.89,Z 783.31,A -85,B 0,C 180,E1 1241.24,E2 1241.24} C_VEL
LIN {X 0,Y 753.917,Z 783.31,A -85,B 0,C 180,E1 1246.041,E2 1246.041} C_VEL
LIN {X 0,Y 753.943,Z 783.31,A -85,B 0,C 180,E1 1250.745,E2 1250.745} C_VEL
LIN {X 0,Y 753.899,Z 783.31,A -85,B 0,C 180,E1 1254.62,E2 1254.62} C_VEL
LIN {X 0,Y 753.971,Z 783.31,A -85,B 0,C 180,E1 1257.208,E2 1257.208} C_VEL
LIN {X 0,Y 752.704,Z 783.31,A -85,B 0,C 180,E1 1257.866,E2 1257.866} C_VEL
LIN {X 0,Y 746.068,Z 783.31,A -85,B 0,C 180,E1 1259.651,E2 1259.651} C_VEL
LIN {X 0,Y 746,Z 783.31,A -85,B 0,C 180,E1 1259.82,E2 1259.82} C_VEL
LIN {X 0,Y 746.214,Z 783.31,A -85,B 0,C 180,E1 1264.654,E2 1264.654} C_VEL
LIN {X 0,Y 746.033,Z 783.31,A -85,B 0,C 180,E1 1269.345,E2 1269.345} C_VEL
LIN {X 0,Y 745.886,Z 783.31,A -85,B 0,C 180,E1 1274.103,E2 1274.103} C_VEL
LIN {X 0,Y 745.976,Z 783.31,A -85,B 0,C 180,E1 1277.732,E2 1277.732} C_VEL
LIN {X 0,Y 745.884,Z 783.31,A -85,B 0,C 180,E1 1281.441,E2 1281.441} C_VEL
LIN {X 0,Y 745.919,Z 783.31,A -85,B 0,C 180,E1 1285.243,E2 1285.243} C_VEL
LIN {X 0,Y 745.927,Z 783.31,A -85,B 0,C 180,E1 1289.168,E2 1289.168} C_VEL
LIN {X 0,Y 745.859,Z 783.31,A -85,B 0,C 180,E1 1293.602,E2 1293.602} C_VEL
LIN {X 0,Y 746,Z 783.31,A -85,B 0,C 180,E1 1297.615,E2 1297.615} C_VEL
LIN {X 0,Y 745.86,Z 783.31,A -85,B 0,C 180,E1 1303.002,E2 1303.002} C_VEL
LIN {X 0,Y 745.856,Z 783.31,A -85,B 0,C 180,E1 1307.903,E2 1307.903} C_VEL
LIN {X 0,Y 746.071,Z 783.31,A -85,B 0,C 180,E1 1312.463,E2 1312.463} C_VEL
LIN {X 0,Y 746.003,Z 783.31,A -85,B 0,C 180,E1 1318.124,E2 1318.124} C_VEL
LIN {X 0,Y 746.179,Z 783.31,A -85,B 0,C 180,E1 1319.712,E2 1319.712} C_VEL
LIN {X 0,Y 748.938,Z 797.846,A -85,B 0,C 180,E1 1320.005,E2 1320.005} C_VEL
LIN {X 0,Y 748.876,Z 863.45,A -85,B 0,C 180,E1 1320.835,E2 1320.835} C_VEL
LIN {X 0,Y 748.484,Z 906.691,A -85,B 0,C 180,E1 1321.859,E2 1321.859} C_VEL
LIN {X 0,Y 748.138,Z 949.117,A -85,B 0,C 180,E1 1323.344,E2 1323.344} C_VEL
LIN {X 0,Y 747.733,Z 991.378,A -85,B 0,C 180,E1 1325.365,E2 1325.365} C_VEL
LIN {X 0,Y 747.222,Z 1031.462,A -85,B 0,C 180,E1 1327.888,E2 1327.888} C_VEL
LIN {X 0,Y 746.838,Z 1066.081,A -85,B 0,C 180,E1 1330.697,E2 1330.697} C_VEL
LIN {X 0,Y 746.5,Z 1095.886,A -85,B 0,C 180,E1 1333.794,E2 1333.794} C_VEL
LIN {X 0,Y 746.261,Z 1119.566,A -85,B 0,C 180,E1 1337.007,E2 1337.007} C_VEL
LIN {X 0,Y 746.248,Z 1135.547,A -85,B 0,C 180,E1 1339.855,E2 1339.855} C_VEL
LIN {X 0,Y 746.177,Z 1148.156,A -85,B 0,C 180,E1 1343.001,E2 1343.001} C_VEL
LIN {X 0,Y 746.214,Z 1155.66,A -85,B 0,C 180,E1 1345.924,E2 1345.924} C_VEL
LIN {X 0,Y 746.231,Z 1159.17,A -85,B 0,C 180,E1 1348.836,E2 1348.836} C_VEL
LIN {X 0,Y 746.318,Z 1158.221,A -85,B 0,C 180,E1 1352.326,E2 1352.326} C_VEL
LIN {X 0,Y 746.271,Z 1151.637,A -85,B 0,C 180,E1 1355.825,E2 1355.825} C_VEL
LIN {X 0,Y 746.301,Z 1140.528,A -85,B 0,C 180,E1 1359.052,E2 1359.052} C_VEL
LIN {X 0,Y 746.382,Z 1122.037,A -85,B 0,C 180,E1 1362.604,E2 1362.604} C_VEL
LIN {X 0,Y 746.482,Z 1098.342,A -85,B 0,C 180,E1 1365.902,E2 1365.902} C_VEL
LIN {X 0,Y 746.778,Z 1071.494,A -85,B 0,C 180,E1 1368.788,E2 1368.788} C_VEL
LIN {X 0,Y 747.153,Z 1039.869,A -85,B 0,C 180,E1 1371.486,E2 1371.486} C_VEL
LIN {X 0,Y 747.615,Z 1002.417,A -85,B 0,C 180,E1 1374.002,E2 1374.002} C_VEL
LIN {X 0,Y 748.081,Z 961.87,A -85,B 0,C 180,E1 1376.107,E2 1376.107} C_VEL
LIN {X 0,Y 748.529,Z 919.336,A -85,B 0,C 180,E1 1377.745,E2 1377.745} C_VEL
LIN {X 0,Y 748.852,Z 879.198,A -85,B 0,C 180,E1 1378.842,E2 1378.842} C_VEL
LIN {X 0,Y 748.953,Z 836.249,A -85,B 0,C 180,E1 1379.57,E2 1379.57} C_VEL
LIN {X 0,Y 748.233,Z 791.999,A -85,B 0,C 180,E1 1380.089,E2 1380.089} C_VEL
LIN {X 0,Y 746.206,Z 783.31,A -85,B 0,C 180,E1 1380.288,E2 1380.288} C_VEL
LIN {X 0,Y 745.853,Z 783.31,A -85,B 0,C 180,E1 1385.666,E2 1385.666} C_VEL
LIN {X 0,Y 745.705,Z 783.31,A -85,B 0,C 180,E1 1389.47,E2 1389.47} C_VEL
LIN {X 0,Y 746.119,Z 783.31,A -85,B 0,C 180,E1 1393.664,E2 1393.664} C_VEL
LIN {X 0,Y 745.705,Z 783.31,A -85,B 0,C 180,E1 1398.744,E2 1398.744} C_VEL
LIN {X 0,Y 745.734,Z 783.31,A -85,B 0,C 180,E1 1402.454,E2 1402.454} C_VEL
LIN {X 0,Y 745.774,Z 783.31,A -85,B 0,C 180,E1 1406.741,E2 1406.741} C_VEL
LIN {X 0,Y 745.817,Z 783.31,A -85,B 0,C 180,E1 1410.873,E2 1410.873} C_VEL
LIN {X 0,Y 746.055,Z 783.31,A -85,B 0,C 180,E1 1414.762,E2 1414.762} C_VEL
LIN {X 0,Y 745.927,Z 783.31,A -85,B 0,C 180,E1 1419.124,E2 1419.124} C_VEL
LIN {X 0,Y 746.004,Z 783.31,A -85,B 0,C 180,E1 1423.486,E2 1423.486} C_VEL
LIN {X 0,Y 745.84,Z 783.31,A -85,B 0,C 180,E1 1428.284,E2 1428.284} C_VEL
LIN {X 0,Y 746.124,Z 783.31,A -85,B 0,C 180,E1 1433.007,E2 1433.007} C_VEL
LIN {X 0,Y 746.111,Z 783.31,A -85,B 0,C 180,E1 1437.677,E2 1437.677} C_VEL
LIN {X 0,Y 745.942,Z 783.31,A -85,B 0,C 180,E1 1442.332,E2 1442.332} C_VEL
LIN {X 0,Y 746.003,Z 783.31,A -85,B 0,C 180,E1 1445.832,E2 1445.832} C_VEL
LIN {X 0,Y 745.923,Z 783.31,A -85,B 0,C 180,E1 1450.537,E2 1450.537} C_VEL
LIN {X 0,Y 746.014,Z 783.31,A -85,B 0,C 180,E1 1455.312,E2 1455.312} C_VEL
LIN {X 0,Y 746.036,Z 783.31,A -85,B 0,C 180,E1 1460.2,E2 1460.2} C_VEL
LIN {X 0,Y 745.859,Z 783.31,A -85,B 0,C 180,E1 1465.254,E2 1465.254} C_VEL
LIN {X 0,Y 745.868,Z 783.31,A -85,B 0,C 180,E1 1469.181,E2 1469.181} C_VEL
LIN {X 0,Y 745.836,Z 783.31,A -85,B 0,C 180,E1 1473.603,E2 1473.603} C_VEL
LIN {X 0,Y 745.986,Z 783.31,A -85,B 0,C 180,E1 1477.617,E2 1477.617} C_VEL
LIN {X 0,Y 746.031,Z 783.31,A -85,B 0,C 180,E1 1483.673,E2 1483.673} C_VEL
LIN {X 0,Y 745.663,Z 783.31,A -85,B 0,C 180,E1 1488.749,E2 1488.749} C_VEL
LIN {X 0,Y 745.735,Z 783.31,A -85,B 0,C 180,E1 1492.446,E2 1492.446} C_VEL
LIN {X 0,Y 745.776,Z 783.31,A -85,B 0,C 180,E1 1496.734,E2 1496.734} C_VEL
LIN {X 0,Y 745.899,Z 783.31,A -85,B 0,C 180,E1 1500.864,E2 1500.864} C_VEL
LIN {X 0,Y 746.152,Z 783.31,A -85,B 0,C 180,E1 1502.931,E2 1502.931} C_VEL
LIN {X 0,Y 748.398,Z 790.146,A -85,B 0,C 180,E1 1503.102,E2 1503.102} C_VEL
LIN {X 0,Y 748.391,Z 860.343,A -85,B 0,C 180,E1 1503.928,E2 1503.928} C_VEL
LIN {X 0,Y 748.193,Z 900.719,A -85,B 0,C 180,E1 1504.833,E2 1504.833} C_VEL
LIN {X 0,Y 747.862,Z 940.365,A -85,B 0,C 180,E1 1506.177,E2 1506.177} C_VEL
LIN {X 0,Y 747.436,Z 978.772,A -85,B 0,C 180,E1 1507.975,E2 1507.975} C_VEL
LIN {X 0,Y 747.015,Z 1015.131,A -85,B 0,C 180,E1 1510.236,E2 1510.236} C_VEL
LIN {X 0,Y 746.705,Z 1047.48,A -85,B 0,C 180,E1 1512.858,E2 1512.858} C_VEL
LIN {X 0,Y 746.453,Z 1073.724,A -85,B 0,C 180,E1 1515.603,E2 1515.603} C_VEL
LIN {X 0,Y 746.344,Z 1095.455,A -85,B 0,C 180,E1 1518.585,E2 1518.585} C_VEL
LIN {X 0,Y 746.225,Z 1112.451,A -85,B 0,C 180,E1 1521.83,E2 1521.83} C_VEL
LIN {X 0,Y 746.255,Z 1122.531,A -85,B 0,C 180,E1 1524.759,E2 1524.759} C_VEL
LIN {X 0,Y 746.273,Z 1128.18,A -85,B 0,C 180,E1 1527.674,E2 1527.674} C_VEL
LIN {X 0,Y 746.322,Z 1129.117,A -85,B 0,C 180,E1 1531.164,E2 1531.164} C_VEL
LIN {X 0,Y 746.284,Z 1125.103,A -85,B 0,C 180,E1 1534.076,E2 1534.076} C_VEL
LIN {X 0,Y 746.304,Z 1115.583,A -85,B 0,C 180,E1 1537.291,E2 1537.291} C_VEL
LIN {X 0,Y 746.368,Z 1101.637,A -85,B 0,C 180,E1 1540.278,E2 1540.278} C_VEL
LIN {X 0,Y 746.516,Z 1080.256,A -85,B 0,C 180,E1 1543.498,E2 1543.498} C_VEL
LIN {X 0,Y 746.701,Z 1053.276,A -85,B 0,C 180,E1 1546.505,E2 1546.505} C_VEL
LIN {X 0,Y 747.01,Z 1021.924,A -85,B 0,C 180,E1 1549.174,E2 1549.174} C_VEL
LIN {X 0,Y 747.32,Z 988.18,A -85,B 0,C 180,E1 1551.405,E2 1551.405} C_VEL
LIN {X 0,Y 747.73,Z 949.477,A -85,B 0,C 180,E1 1553.355,E2 1553.355} C_VEL
LIN {X 0,Y 748.078,Z 907.951,A -85,B 0,C 180,E1 1554.873,E2 1554.873} C_VEL
LIN {X 0,Y 748.329,Z 865.485,A -85,B 0,C 180,E1 1555.899,E2 1555.899} C_VEL
LIN {X 0,Y 748.165,Z 797.527,A -85,B 0,C 180,E1 1556.739,E2 1556.739} C_VEL
LIN {X 0,Y 747.126,Z 786.819,A -85,B 0,C 180,E1 1556.892,E2 1556.892} C_VEL
LIN {X 0,Y 746.259,Z 783.31,A -85,B 0,C 180,E1 1556.996,E2 1556.996} C_VEL
LIN {X 0,Y 746.038,Z 783.31,A -85,B 0,C 180,E1 1561.875,E2 1561.875} C_VEL
LIN {X 0,Y 745.993,Z 783.31,A -85,B 0,C 180,E1 1567.616,E2 1567.616} C_VEL
LIN {X 0,Y 746.043,Z 783.31,A -85,B 0,C 180,E1 1573.672,E2 1573.672} C_VEL
LIN {X 0,Y 745.661,Z 783.31,A -85,B 0,C 180,E1 1578.751,E2 1578.751} C_VEL
LIN {X 0,Y 745.708,Z 783.31,A -85,B 0,C 180,E1 1582.441,E2 1582.441} C_VEL
LIN {X 0,Y 745.757,Z 783.31,A -85,B 0,C 180,E1 1586.73,E2 1586.73} C_VEL
LIN {X 0,Y 745.817,Z 783.31,A -85,B 0,C 180,E1 1590.878,E2 1590.878} C_VEL
LIN {X 0,Y 746.005,Z 783.31,A -85,B 0,C 180,E1 1594.751,E2 1594.751} C_VEL
LIN {X 0,Y 745.88,Z 783.31,A -85,B 0,C 180,E1 1599.139,E2 1599.139} C_VEL
LIN {X 0,Y 745.999,Z 783.31,A -85,B 0,C 180,E1 1603.477,E2 1603.477} C_VEL
LIN {X 0,Y 745.881,Z 783.31,A -85,B 0,C 180,E1 1608.276,E2 1608.276} C_VEL
LIN {X 0,Y 746.191,Z 783.31,A -85,B 0,C 180,E1 1612.998,E2 1612.998} C_VEL
LIN {X 0,Y 746.113,Z 783.31,A -85,B 0,C 180,E1 1617.668,E2 1617.668} C_VEL
LIN {X 0,Y 746,Z 783.31,A -85,B 0,C 180,E1 1619.82,E2 1619.82} C_VEL
LIN {X 0,Y 743.556,Z 783.31,A -85,B 0,C 180,E1 1620.811,E2 1620.811} C_VEL
LIN {X 0,Y 738.15,Z 783.31,A -85,B 0,C 180,E1 1622.29,E2 1622.29} C_VEL
LIN {X 0,Y 738.044,Z 783.31,A -85,B 0,C 180,E1 1622.461,E2 1622.461} C_VEL
LIN {X 0,Y 738.098,Z 783.31,A -85,B 0,C 180,E1 1625.886,E2 1625.886} C_VEL
LIN {X 0,Y 738.028,Z 783.31,A -85,B 0,C 180,E1 1630.642,E2 1630.642} C_VEL
LIN {X 0,Y 738.165,Z 783.31,A -85,B 0,C 180,E1 1635.47,E2 1635.47} C_VEL
LIN {X 0,Y 738.148,Z 783.31,A -85,B 0,C 180,E1 1640.416,E2 1640.416} C_VEL
LIN {X 0,Y 737.987,Z 783.31,A -85,B 0,C 180,E1 1645.533,E2 1645.533} C_VEL
LIN {X 0,Y 737.938,Z 783.31,A -85,B 0,C 180,E1 1650.415,E2 1650.415} C_VEL
LIN {X 0,Y 737.87,Z 783.31,A -85,B 0,C 180,E1 1655.088,E2 1655.088} C_VEL
LIN {X 0,Y 737.73,Z 783.31,A -85,B 0,C 180,E1 1659.535,E2 1659.535} C_VEL
LIN {X 0,Y 737.792,Z 783.31,A -85,B 0,C 180,E1 1664.045,E2 1664.045} C_VEL
LIN {X 0,Y 737.81,Z 783.31,A -85,B 0,C 180,E1 1668.916,E2 1668.916} C_VEL
LIN {X 0,Y 738.066,Z 783.31,A -85,B 0,C 180,E1 1673.462,E2 1673.462} C_VEL
LIN {X 0,Y 738.191,Z 783.31,A -85,B 0,C 180,E1 1679.126,E2 1679.126} C_VEL
LIN {X 0,Y 738.223,Z 783.816,A -85,B 0,C 180,E1 1679.369,E2 1679.369} C_VEL
LIN {X 0,Y 742.096,Z 797.067,A -85,B 0,C 180,E1 1679.691,E2 1679.691} C_VEL
LIN {X 0,Y 741.973,Z 863.452,A -85,B 0,C 180,E1 1680.537,E2 1680.537} C_VEL
LIN {X 0,Y 741.422,Z 907.359,A -85,B 0,C 180,E1 1681.587,E2 1681.587} C_VEL
LIN {X 0,Y 740.922,Z 950.262,A -85,B 0,C 180,E1 1683.113,E2 1683.113} C_VEL
LIN {X 0,Y 740.339,Z 992.112,A -85,B 0,C 180,E1 1685.145,E2 1685.145} C_VEL
LIN {X 0,Y 739.725,Z 1030.776,A -85,B 0,C 180,E1 1687.601,E2 1687.601} C_VEL
LIN {X 0,Y 739.167,Z 1064.894,A -85,B 0,C 180,E1 1690.377,E2 1690.377} C_VEL
LIN {X 0,Y 738.71,Z 1094.564,A -85,B 0,C 180,E1 1693.465,E2 1693.465} C_VEL
LIN {X 0,Y 738.438,Z 1118.175,A -85,B 0,C 180,E1 1696.653,E2 1696.653} C_VEL
LIN {X 0,Y 738.366,Z 1135.515,A -85,B 0,C 180,E1 1699.738,E2 1699.738} C_VEL
LIN {X 0,Y 738.287,Z 1148.156,A -85,B 0,C 180,E1 1702.926,E2 1702.926} C_VEL
LIN {X 0,Y 738.316,Z 1155.66,A -85,B 0,C 180,E1 1705.88,E2 1705.88} C_VEL
LIN {X 0,Y 738.33,Z 1159.17,A -85,B 0,C 180,E1 1708.823,E2 1708.823} C_VEL
LIN {X 0,Y 738.427,Z 1158.221,A -85,B 0,C 180,E1 1712.351,E2 1712.351} C_VEL
LIN {X 0,Y 738.398,Z 1151.637,A -85,B 0,C 180,E1 1715.888,E2 1715.888} C_VEL
LIN {X 0,Y 738.403,Z 1140.528,A -85,B 0,C 180,E1 1719.149,E2 1719.149} C_VEL
LIN {X 0,Y 738.513,Z 1122.038,A -85,B 0,C 180,E1 1722.74,E2 1722.74} C_VEL
LIN {X 0,Y 738.69,Z 1098.344,A -85,B 0,C 180,E1 1726.074,E2 1726.074} C_VEL
LIN {X 0,Y 739.05,Z 1071.495,A -85,B 0,C 180,E1 1728.992,E2 1728.992} C_VEL
LIN {X 0,Y 739.57,Z 1039.908,A -85,B 0,C 180,E1 1731.715,E2 1731.715} C_VEL
LIN {X 0,Y 740.189,Z 1002.42,A -85,B 0,C 180,E1 1734.258,E2 1734.258} C_VEL
LIN {X 0,Y 740.823,Z 962.106,A -85,B 0,C 180,E1 1736.371,E2 1736.371} C_VEL
LIN {X 0,Y 741.44,Z 919.34,A -85,B 0,C 180,E1 1738.034,E2 1738.034} C_VEL
LIN {X 0,Y 741.912,Z 878.289,A -85,B 0,C 180,E1 1739.157,E2 1739.157} C_VEL
LIN {X 0,Y 742.088,Z 834.282,A -85,B 0,C 180,E1 1739.897,E2 1739.897} C_VEL
LIN {X 0,Y 741.413,Z 793.633,A -85,B 0,C 180,E1 1740.377,E2 1740.377} C_VEL
LIN {X 0,Y 738.266,Z 783.31,A -85,B 0,C 180,E1 1740.659,E2 1740.659} C_VEL
LIN {X 0,Y 738.029,Z 783.31,A -85,B 0,C 180,E1 1746.537,E2 1746.537} C_VEL
LIN {X 0,Y 738.077,Z 783.31,A -85,B 0,C 180,E1 1752.364,E2 1752.364} C_VEL
LIN {X 0,Y 738.018,Z 783.31,A -85,B 0,C 180,E1 1755.934,E2 1755.934} C_VEL
LIN {X 0,Y 737.909,Z 783.31,A -85,B 0,C 180,E1 1761.283,E2 1761.283} C_VEL
LIN {X 0,Y 737.897,Z 783.31,A -85,B 0,C 180,E1 1766.339,E2 1766.339} C_VEL
LIN {X 0,Y 737.924,Z 783.31,A -85,B 0,C 180,E1 1770.484,E2 1770.484} C_VEL
LIN {X 0,Y 738.171,Z 783.31,A -85,B 0,C 180,E1 1774.571,E2 1774.571} C_VEL
LIN {X 0,Y 738.123,Z 783.31,A -85,B 0,C 180,E1 1778.323,E2 1778.323} C_VEL
LIN {X 0,Y 738.111,Z 783.31,A -85,B 0,C 180,E1 1783.305,E2 1783.305} C_VEL
LIN {X 0,Y 737.932,Z 783.31,A -85,B 0,C 180,E1 1788.157,E2 1788.157} C_VEL
LIN {X 0,Y 738.199,Z 783.31,A -85,B 0,C 180,E1 1792.931,E2 1792.931} C_VEL
LIN {X 0,Y 738.209,Z 783.31,A -85,B 0,C 180,E1 1797.652,E2 1797.652} C_VEL
LIN {X 0,Y 738.051,Z 783.31,A -85,B 0,C 180,E1 1802.357,E2 1802.357} C_VEL
LIN {X 0,Y 738.091,Z 783.31,A -85,B 0,C 180,E1 1805.895,E2 1805.895} C_VEL
LIN {X 0,Y 738.041,Z 783.31,A -85,B 0,C 180,E1 1810.651,E2 1810.651} C_VEL
LIN {X 0,Y 738.105,Z 783.31,A -85,B 0,C 180,E1 1815.481,E2 1815.481} C_VEL
LIN {X 0,Y 738.094,Z 783.31,A -85,B 0,C 180,E1 1820.427,E2 1820.427} C_VEL
LIN {X 0,Y 737.922,Z 783.31,A -85,B 0,C 180,E1 1825.545,E2 1825.545} C_VEL
LIN {X 0,Y 737.892,Z 783.31,A -85,B 0,C 180,E1 1830.413,E2 1830.413} C_VEL
LIN {X 0,Y 737.854,Z 783.31,A -85,B 0,C 180,E1 1835.099,E2 1835.099} C_VEL
LIN {X 0,Y 737.732,Z 783.31,A -85,B 0,C 180,E1 1839.546,E2 1839.546} C_VEL
LIN {X 0,Y 738.135,Z 783.31,A -85,B 0,C 180,E1 1844.261,E2 1844.261} C_VEL
LIN {X 0,Y 737.91,Z 783.31,A -85,B 0,C 180,E1 1849.441,E2 1849.441} C_VEL
LIN {X 0,Y 737.944,Z 783.31,A -85,B 0,C 180,E1 1854.909,E2 1854.909} C_VEL
LIN {X 0,Y 738.106,Z 783.31,A -85,B 0,C 180,E1 1859.56,E2 1859.56} C_VEL
LIN {X 0,Y 738.201,Z 783.653,A -85,B 0,C 180,E1 1862.631,E2 1862.631} C_VEL
LIN {X 0,Y 741.385,Z 794.392,A -85,B 0,C 180,E1 1862.873,E2 1862.873} C_VEL
LIN {X 0,Y 741.28,Z 862.028,A -85,B 0,C 180,E1 1863.687,E2 1863.687} C_VEL
LIN {X 0,Y 740.992,Z 903.715,A -85,B 0,C 180,E1 1864.659,E2 1864.659} C_VEL
LIN {X 0,Y 740.481,Z 942.251,A -85,B 0,C 180,E1 1866.005,E2 1866.005} C_VEL
LIN {X 0,Y 739.938,Z 980.153,A -85,B 0,C 180,E1 1867.82,E2 1867.82} C_VEL
LIN {X 0,Y 739.448,Z 1014.813,A -85,B 0,C 180,E1 1870.002,E2 1870.002} C_VEL
LIN {X 0,Y 738.958,Z 1047.084,A -85,B 0,C 180,E1 1872.636,E2 1872.636} C_VEL
LIN {X 0,Y 738.664,Z 1073.736,A -85,B 0,C 180,E1 1875.45,E2 1875.45} C_VEL
LIN {X 0,Y 738.508,Z 1095.453,A -85,B 0,C 180,E1 1878.462,E2 1878.462} C_VEL
LIN {X 0,Y 738.353,Z 1112.448,A -85,B 0,C 180,E1 1881.742,E2 1881.742} C_VEL
LIN {X 0,Y 738.349,Z 1122.768,A -85,B 0,C 180,E1 1884.793,E2 1884.793} C_VEL
LIN {X 0,Y 738.393,Z 1128.18,A -85,B 0,C 180,E1 1887.649,E2 1887.649} C_VEL
LIN {X 0,Y 738.42,Z 1129.118,A -85,B 0,C 180,E1 1891.177,E2 1891.177} C_VEL
LIN {X 0,Y 738.372,Z 1125.105,A -85,B 0,C 180,E1 1894.12,E2 1894.12} C_VEL
LIN {X 0,Y 738.431,Z 1115.585,A -85,B 0,C 180,E1 1897.369,E2 1897.369} C_VEL
LIN {X 0,Y 738.472,Z 1101.271,A -85,B 0,C 180,E1 1900.453,E2 1900.453} C_VEL
LIN {X 0,Y 738.655,Z 1080.254,A -85,B 0,C 180,E1 1903.645,E2 1903.645} C_VEL
LIN {X 0,Y 738.953,Z 1053.28,A -85,B 0,C 180,E1 1906.683,E2 1906.683} C_VEL
LIN {X 0,Y 739.347,Z 1022.04,A -85,B 0,C 180,E1 1909.373,E2 1909.373} C_VEL
LIN {X 0,Y 739.828,Z 988.192,A -85,B 0,C 180,E1 1911.633,E2 1911.633} C_VEL
LIN {X 0,Y 740.402,Z 949.507,A -85,B 0,C 180,E1 1913.599,E2 1913.599} C_VEL
LIN {X 0,Y 740.852,Z 909.216,A -85,B 0,C 180,E1 1915.096,E2 1915.096} C_VEL
LIN {X 0,Y 741.254,Z 864.49,A -85,B 0,C 180,E1 1916.183,E2 1916.183} C_VEL
LIN {X 0,Y 740.941,Z 790.954,A -85,B 0,C 180,E1 1917.091,E2 1917.091} C_VEL
LIN {X 0,Y 738.336,Z 783.31,A -85,B 0,C 180,E1 1917.334,E2 1917.334} C_VEL
LIN {X 0,Y 738.036,Z 783.31,A -85,B 0,C 180,E1 1922.678,E2 1922.678} C_VEL
LIN {X 0,Y 737.967,Z 783.31,A -85,B 0,C 180,E1 1928.022,E2 1928.022} C_VEL
LIN {X 0,Y 738.14,Z 783.31,A -85,B 0,C 180,E1 1934.074,E2 1934.074} C_VEL
LIN {X 0,Y 737.897,Z 783.31,A -85,B 0,C 180,E1 1939.443,E2 1939.443} C_VEL
LIN {X 0,Y 737.927,Z 783.31,A -85,B 0,C 180,E1 1944.905,E2 1944.905} C_VEL
LIN {X 0,Y 738.05,Z 783.31,A -85,B 0,C 180,E1 1949.57,E2 1949.57} C_VEL
LIN {X 0,Y 738.11,Z 783.31,A -85,B 0,C 180,E1 1954.586,E2 1954.586} C_VEL
LIN {X 0,Y 738.071,Z 783.31,A -85,B 0,C 180,E1 1958.312,E2 1958.312} C_VEL
LIN {X 0,Y 738.11,Z 783.31,A -85,B 0,C 180,E1 1963.295,E2 1963.295} C_VEL
LIN {X 0,Y 737.969,Z 783.31,A -85,B 0,C 180,E1 1968.149,E2 1968.149} C_VEL
LIN {X 0,Y 738.268,Z 783.31,A -85,B 0,C 180,E1 1972.923,E2 1972.923} C_VEL
LIN {X 0,Y 738.213,Z 783.31,A -85,B 0,C 180,E1 1977.643,E2 1977.643} C_VEL
LIN {X 0,Y 738.044,Z 783.31,A -85,B 0,C 180,E1 1982.461,E2 1982.461} C_VEL
LIN {X 0,Y 734.233,Z 783.31,A -85,B 0,C 180,E1 1983.787,E2 1983.787} C_VEL
LIN {X 0,Y 730.307,Z 783.31,A -85,B 0,C 180,E1 1985.126,E2 1985.126} C_VEL
LIN {X 0,Y 730.19,Z 783.31,A -85,B 0,C 180,E1 1989.55,E2 1989.55} C_VEL
LIN {X 0,Y 730.108,Z 783.31,A -85,B 0,C 180,E1 1994.414,E2 1994.414} C_VEL
LIN {X 0,Y 730.24,Z 783.31,A -85,B 0,C 180,E1 1999.382,E2 1999.382} C_VEL
LIN {X 0,Y 730.182,Z 783.31,A -85,B 0,C 180,E1 2004.513,E2 2004.513} C_VEL
LIN {X 0,Y 730.033,Z 783.31,A -85,B 0,C 180,E1 2009.867,E2 2009.867} C_VEL
LIN {X 0,Y 729.993,Z 783.31,A -85,B 0,C 180,E1 2014.075,E2 2014.075} C_VEL
LIN {X 0,Y 729.959,Z 783.31,A -85,B 0,C 180,E1 2018.504,E2 2018.504} C_VEL
LIN {X 0,Y 729.917,Z 783.31,A -85,B 0,C 180,E1 2023.402,E2 2023.402} C_VEL
LIN {X 0,Y 729.952,Z 783.31,A -85,B 0,C 180,E1 2028.376,E2 2028.376} C_VEL
LIN {X 0,Y 730.157,Z 783.31,A -85,B 0,C 180,E1 2033.001,E2 2033.001} C_VEL
LIN {X 0,Y 730.179,Z 783.31,A -85,B 0,C 180,E1 2038.279,E2 2038.279} C_VEL
LIN {X 0,Y 730.262,Z 783.31,A -85,B 0,C 180,E1 2038.973,E2 2038.973} C_VEL
LIN {X 0,Y 735.186,Z 797.562,A -85,B 0,C 180,E1 2039.382,E2 2039.382} C_VEL
LIN {X 0,Y 735.082,Z 864.104,A -85,B 0,C 180,E1 2040.245,E2 2040.245} C_VEL
LIN {X 0,Y 734.392,Z 909.487,A -85,B 0,C 180,E1 2041.354,E2 2041.354} C_VEL
LIN {X 0,Y 733.742,Z 951.031,A -85,B 0,C 180,E1 2042.862,E2 2042.862} C_VEL
LIN {X 0,Y 732.974,Z 991.545,A -85,B 0,C 180,E1 2044.845,E2 2044.845} C_VEL
LIN {X 0,Y 732.192,Z 1030.039,A -85,B 0,C 180,E1 2047.304,E2 2047.304} C_VEL
LIN {X 0,Y 731.522,Z 1065.223,A -85,B 0,C 180,E1 2050.193,E2 2050.193} C_VEL
LIN {X 0,Y 730.917,Z 1095.886,A -85,B 0,C 180,E1 2053.438,E2 2053.438} C_VEL
LIN {X 0,Y 730.581,Z 1120.142,A -85,B 0,C 180,E1 2056.812,E2 2056.812} C_VEL
LIN {X 0,Y 730.489,Z 1136.671,A -85,B 0,C 180,E1 2059.886,E2 2059.886} C_VEL
LIN {X 0,Y 730.404,Z 1148.157,A -85,B 0,C 180,E1 2062.849,E2 2062.849} C_VEL
LIN {X 0,Y 730.429,Z 1155.66,A -85,B 0,C 180,E1 2065.836,E2 2065.836} C_VEL
LIN {X 0,Y 730.428,Z 1159.17,A -85,B 0,C 180,E1 2068.81,E2 2068.81} C_VEL
LIN {X 0,Y 730.522,Z 1158.222,A -85,B 0,C 180,E1 2072.376,E2 2072.376} C_VEL
LIN {X 0,Y 730.492,Z 1151.638,A -85,B 0,C 180,E1 2075.952,E2 2075.952} C_VEL
LIN {X 0,Y 730.5,Z 1140.527,A -85,B 0,C 180,E1 2079.249,E2 2079.249} C_VEL
LIN {X 0,Y 730.656,Z 1122.942,A -85,B 0,C 180,E1 2082.723,E2 2082.723} C_VEL
LIN {X 0,Y 730.891,Z 1100.777,A -85,B 0,C 180,E1 2085.942,E2 2085.942} C_VEL
LIN {X 0,Y 731.343,Z 1073.107,A -85,B 0,C 180,E1 2089.043,E2 2089.043} C_VEL
LIN {X 0,Y 731.973,Z 1040.917,A -85,B 0,C 180,E1 2091.875,E2 2091.875} C_VEL
LIN {X 0,Y 732.767,Z 1004,A -85,B 0,C 180,E1 2094.427,E2 2094.427} C_VEL
LIN {X 0,Y 733.6,Z 962.662,A -85,B 0,C 180,E1 2096.624,E2 2096.624} C_VEL
LIN {X 0,Y 734.362,Z 920.439,A -85,B 0,C 180,E1 2098.29,E2 2098.29} C_VEL
LIN {X 0,Y 734.974,Z 878.89,A -85,B 0,C 180,E1 2099.447,E2 2099.447} C_VEL
LIN {X 0,Y 735.24,Z 835.438,A -85,B 0,C 180,E1 2100.189,E2 2100.189} C_VEL
LIN {X 0,Y 734.632,Z 795.264,A -85,B 0,C 180,E1 2100.67,E2 2100.67} C_VEL
LIN {X 0,Y 730.316,Z 783.31,A -85,B 0,C 180,E1 2101.065,E2 2101.065} C_VEL
LIN {X 0,Y 730.14,Z 783.31,A -85,B 0,C 180,E1 2106.997,E2 2106.997} C_VEL
LIN {X 0,Y 730.031,Z 783.31,A -85,B 0,C 180,E1 2111.667,E2 2111.667} C_VEL
LIN {X 0,Y 730.149,Z 783.31,A -85,B 0,C 180,E1 2115.138,E2 2115.138} C_VEL
LIN {X 0,Y 730.078,Z 783.31,A -85,B 0,C 180,E1 2120.162,E2 2120.162} C_VEL
LIN {X 0,Y 729.965,Z 783.31,A -85,B 0,C 180,E1 2124.475,E2 2124.475} C_VEL
LIN {X 0,Y 730.099,Z 783.31,A -85,B 0,C 180,E1 2128.755,E2 2128.755} C_VEL
LIN {X 0,Y 730.219,Z 783.31,A -85,B 0,C 180,E1 2134.175,E2 2134.175} C_VEL
LIN {X 0,Y 730.093,Z 783.31,A -85,B 0,C 180,E1 2139.046,E2 2139.046} C_VEL
LIN {X 0,Y 730.192,Z 783.31,A -85,B 0,C 180,E1 2143.118,E2 2143.118} C_VEL
LIN {X 0,Y 730.017,Z 783.31,A -85,B 0,C 180,E1 2148.027,E2 2148.027} C_VEL
LIN {X 0,Y 730.303,Z 783.31,A -85,B 0,C 180,E1 2152.854,E2 2152.854} C_VEL
LIN {X 0,Y 730.305,Z 783.31,A -85,B 0,C 180,E1 2157.627,E2 2157.627} C_VEL
LIN {X 0,Y 730.149,Z 783.31,A -85,B 0,C 180,E1 2162.383,E2 2162.383} C_VEL
LIN {X 0,Y 730.211,Z 783.31,A -85,B 0,C 180,E1 2165.959,E2 2165.959} C_VEL
LIN {X 0,Y 730.139,Z 783.31,A -85,B 0,C 180,E1 2170.768,E2 2170.768} C_VEL
LIN {X 0,Y 730.189,Z 783.31,A -85,B 0,C 180,E1 2175.653,E2 2175.653} C_VEL
LIN {X 0,Y 730.092,Z 783.31,A -85,B 0,C 180,E1 2180.954,E2 2180.954} C_VEL
LIN {X 0,Y 729.992,Z 783.31,A -85,B 0,C 180,E1 2185.843,E2 2185.843} C_VEL
LIN {X 0,Y 729.993,Z 783.31,A -85,B 0,C 180,E1 2189.879,E2 2189.879} C_VEL
LIN {X 0,Y 729.974,Z 783.31,A -85,B 0,C 180,E1 2194.087,E2 2194.087} C_VEL
LIN {X 0,Y 729.949,Z 783.31,A -85,B 0,C 180,E1 2198.516,E2 2198.516} C_VEL
LIN {X 0,Y 730.138,Z 783.31,A -85,B 0,C 180,E1 2203.424,E2 2203.424} C_VEL
LIN {X 0,Y 729.845,Z 783.31,A -85,B 0,C 180,E1 2208.371,E2 2208.371} C_VEL
LIN {X 0,Y 729.911,Z 783.31,A -85,B 0,C 180,E1 2212.989,E2 2212.989} C_VEL
LIN {X 0,Y 730.052,Z 783.31,A -85,B 0,C 180,E1 2218.312,E2 2218.312} C_VEL
LIN {X 0,Y 730.204,Z 783.567,A -85,B 0,C 180,E1 2222.306,E2 2222.306} C_VEL
LIN {X 0,Y 734.357,Z 794.564,A -85,B 0,C 180,E1 2222.594,E2 2222.594} C_VEL
LIN {X 0,Y 734.182,Z 863.566,A -85,B 0,C 180,E1 2223.439,E2 2223.439} C_VEL
LIN {X 0,Y 733.808,Z 905.228,A -85,B 0,C 180,E1 2224.438,E2 2224.438} C_VEL
LIN {X 0,Y 733.124,Z 944.123,A -85,B 0,C 180,E1 2225.83,E2 2225.83} C_VEL
LIN {X 0,Y 732.439,Z 982.43,A -85,B 0,C 180,E1 2227.712,E2 2227.712} C_VEL
LIN {X 0,Y 731.784,Z 1017.234,A -85,B 0,C 180,E1 2229.966,E2 2229.966} C_VEL
LIN {X 0,Y 731.246,Z 1047.533,A -85,B 0,C 180,E1 2232.49,E2 2232.49} C_VEL
LIN {X 0,Y 730.877,Z 1073.953,A -85,B 0,C 180,E1 2235.319,E2 2235.319} C_VEL
LIN {X 0,Y 730.658,Z 1095.45,A -85,B 0,C 180,E1 2238.336,E2 2238.336} C_VEL
LIN {X 0,Y 730.488,Z 1112.446,A -85,B 0,C 180,E1 2241.653,E2 2241.653} C_VEL
LIN {X 0,Y 730.477,Z 1122.481,A -85,B 0,C 180,E1 2244.627,E2 2244.627} C_VEL
LIN {X 0,Y 730.487,Z 1128.179,A -85,B 0,C 180,E1 2247.624,E2 2247.624} C_VEL
LIN {X 0,Y 730.518,Z 1129.118,A -85,B 0,C 180,E1 2251.189,E2 2251.189} C_VEL
LIN {X 0,Y 730.474,Z 1125.107,A -85,B 0,C 180,E1 2254.164,E2 2254.164} C_VEL
LIN {X 0,Y 730.547,Z 1115.587,A -85,B 0,C 180,E1 2257.449,E2 2257.449} C_VEL
LIN {X 0,Y 730.6,Z 1101.977,A -85,B 0,C 180,E1 2260.441,E2 2260.441} C_VEL
LIN {X 0,Y 730.804,Z 1080.257,A -85,B 0,C 180,E1 2263.795,E2 2263.795} C_VEL
LIN {X 0,Y 731.196,Z 1053.284,A -85,B 0,C 180,E1 2266.865,E2 2266.865} C_VEL
LIN {X 0,Y 731.712,Z 1022.048,A -85,B 0,C 180,E1 2269.583,E2 2269.583} C_VEL
LIN {X 0,Y 732.331,Z 986.981,A -85,B 0,C 180,E1 2271.937,E2 2271.937} C_VEL
LIN {X 0,Y 733.064,Z 949.51,A -85,B 0,C 180,E1 2273.851,E2 2273.851} C_VEL
LIN {X 0,Y 733.708,Z 908.293,A -85,B 0,C 180,E1 2275.385,E2 2275.385} C_VEL
LIN {X 0,Y 734.169,Z 863.806,A -85,B 0,C 180,E1 2276.467,E2 2276.467} C_VEL
LIN {X 0,Y 733.63,Z 792.467,A -85,B 0,C 180,E1 2277.368,E2 2277.368} C_VEL
LIN {X 0,Y 730.398,Z 783.31,A -85,B 0,C 180,E1 2277.645,E2 2277.645} C_VEL
LIN {X 0,Y 730.151,Z 783.31,A -85,B 0,C 180,E1 2282.653,E2 2282.653} C_VEL
LIN {X 0,Y 730.059,Z 783.31,A -85,B 0,C 180,E1 2287.94,E2 2287.94} C_VEL
LIN {X 0,Y 730.151,Z 783.31,A -85,B 0,C 180,E1 2293.422,E2 2293.422} C_VEL
LIN {X 0,Y 729.866,Z 783.31,A -85,B 0,C 180,E1 2298.37,E2 2298.37} C_VEL
LIN {X 0,Y 729.887,Z 783.31,A -85,B 0,C 180,E1 2302.985,E2 2302.985} C_VEL
LIN {X 0,Y 729.969,Z 783.31,A -85,B 0,C 180,E1 2307.337,E2 2307.337} C_VEL
LIN {X 0,Y 729.982,Z 783.31,A -85,B 0,C 180,E1 2311.483,E2 2311.483} C_VEL
LIN {X 0,Y 730.113,Z 783.31,A -85,B 0,C 180,E1 2315.941,E2 2315.941} C_VEL
LIN {X 0,Y 730.108,Z 783.31,A -85,B 0,C 180,E1 2320.604,E2 2320.604} C_VEL
LIN {X 0,Y 730.164,Z 783.31,A -85,B 0,C 180,E1 2325.578,E2 2325.578} C_VEL
LIN {X 0,Y 730.285,Z 783.31,A -85,B 0,C 180,E1 2330.442,E2 2330.442} C_VEL
LIN {X 0,Y 730.144,Z 783.31,A -85,B 0,C 180,E1 2335.235,E2 2335.235} C_VEL
LIN {X 0,Y 730.238,Z 783.31,A -85,B 0,C 180,E1 2339.996,E2 2339.996} C_VEL
LIN {X 0,Y 730.307,Z 783.31,A -85,B 0,C 180,E1 2345.126,E2 2345.126} C_VEL
LIN {X 0,Y 726.176,Z 783.31,A -85,B 0,C 180,E1 2346.46,E2 2346.46} C_VEL
LIN {X 0,Y 722.275,Z 783.31,A -85,B 0,C 180,E1 2347.809,E2 2347.809} C_VEL
LIN {X 0,Y 722.282,Z 783.31,A -85,B 0,C 180,E1 2353.335,E2 2353.335} C_VEL
LIN {X 0,Y 722.251,Z 783.31,A -85,B 0,C 180,E1 2358.335,E2 2358.335} C_VEL
LIN {X 0,Y 722.24,Z 783.31,A -85,B 0,C 180,E1 2363.483,E2 2363.483} C_VEL
LIN {X 0,Y 722.179,Z 783.31,A -85,B 0,C 180,E1 2368.844,E2 2368.844} C_VEL
LIN {X 0,Y 722.186,Z 783.31,A -85,B 0,C 180,E1 2373.049,E2 2373.049} C_VEL
LIN {X 0,Y 722.156,Z 783.31,A -85,B 0,C 180,E1 2377.468,E2 2377.468} C_VEL
LIN {X 0,Y 722,Z 783.31,A -85,B 0,C 180,E1 2382.734,E2 2382.734} C_VEL
LIN {X 0,Y 722.008,Z 783.31,A -85,B 0,C 180,E1 2387.813,E2 2387.813} C_VEL
LIN {X 0,Y 722.264,Z 783.31,A -85,B 0,C 180,E1 2392.846,E2 2392.846} C_VEL
LIN {X 0,Y 722.314,Z 783.31,A -85,B 0,C 180,E1 2398.597,E2 2398.597} C_VEL
LIN {X 0,Y 728.452,Z 799.863,A -85,B 0,C 180,E1 2399.094,E2 2399.094} C_VEL
LIN {X 0,Y 728.229,Z 864.105,A -85,B 0,C 180,E1 2399.936,E2 2399.936} C_VEL
LIN {X 0,Y 727.377,Z 908.195,A -85,B 0,C 180,E1 2401.012,E2 2401.012} C_VEL
LIN {X 0,Y 726.603,Z 949.688,A -85,B 0,C 180,E1 2402.514,E2 2402.514} C_VEL
LIN {X 0,Y 725.657,Z 991.531,A -85,B 0,C 180,E1 2404.573,E2 2404.573} C_VEL
LIN {X 0,Y 724.655,Z 1030.774,A -85,B 0,C 180,E1 2407.109,E2 2407.109} C_VEL
LIN {X 0,Y 723.85,Z 1065.003,A -85,B 0,C 180,E1 2409.954,E2 2409.954} C_VEL
LIN {X 0,Y 723.161,Z 1094.56,A -85,B 0,C 180,E1 2413.099,E2 2413.099} C_VEL
LIN {X 0,Y 722.831,Z 1116.209,A -85,B 0,C 180,E1 2416.05,E2 2416.05} C_VEL
LIN {X 0,Y 722.663,Z 1135.077,A -85,B 0,C 180,E1 2419.415,E2 2419.415} C_VEL
LIN {X 0,Y 722.518,Z 1148.157,A -85,B 0,C 180,E1 2422.771,E2 2422.771} C_VEL
LIN {X 0,Y 722.556,Z 1155.661,A -85,B 0,C 180,E1 2425.79,E2 2425.79} C_VEL
LIN {X 0,Y 722.526,Z 1159.169,A -85,B 0,C 180,E1 2428.797,E2 2428.797} C_VEL
LIN {X 0,Y 722.635,Z 1158.221,A -85,B 0,C 180,E1 2432.402,E2 2432.402} C_VEL
LIN {X 0,Y 722.58,Z 1151.638,A -85,B 0,C 180,E1 2436.017,E2 2436.017} C_VEL
LIN {X 0,Y 722.635,Z 1140.527,A -85,B 0,C 180,E1 2439.351,E2 2439.351} C_VEL
LIN {X 0,Y 722.804,Z 1122.102,A -85,B 0,C 180,E1 2443.011,E2 2443.011} C_VEL
LIN {X 0,Y 723.129,Z 1099.563,A -85,B 0,C 180,E1 2446.274,E2 2446.274} C_VEL
LIN {X 0,Y 723.634,Z 1073.107,A -85,B 0,C 180,E1 2449.254,E2 2449.254} C_VEL
LIN {X 0,Y 724.432,Z 1040.918,A -85,B 0,C 180,E1 2452.114,E2 2452.114} C_VEL
LIN {X 0,Y 725.366,Z 1004.001,A -85,B 0,C 180,E1 2454.692,E2 2454.692} C_VEL
LIN {X 0,Y 726.416,Z 962.657,A -85,B 0,C 180,E1 2456.909,E2 2456.909} C_VEL
LIN {X 0,Y 727.317,Z 921.007,A -85,B 0,C 180,E1 2458.57,E2 2458.57} C_VEL
LIN {X 0,Y 728.038,Z 880.565,A -85,B 0,C 180,E1 2459.719,E2 2459.719} C_VEL
LIN {X 0,Y 728.403,Z 835.78,A -85,B 0,C 180,E1 2460.498,E2 2460.498} C_VEL
LIN {X 0,Y 727.764,Z 796.464,A -85,B 0,C 180,E1 2460.977,E2 2460.977} C_VEL
LIN {X 0,Y 722.397,Z 783.31,A -85,B 0,C 180,E1 2461.428,E2 2461.428} C_VEL
LIN {X 0,Y 722.24,Z 783.31,A -85,B 0,C 180,E1 2467.471,E2 2467.471} C_VEL
LIN {X 0,Y 722.204,Z 783.31,A -85,B 0,C 180,E1 2472.765,E2 2472.765} C_VEL
LIN {X 0,Y 721.948,Z 783.31,A -85,B 0,C 180,E1 2477.821,E2 2477.821} C_VEL
LIN {X 0,Y 722.032,Z 783.31,A -85,B 0,C 180,E1 2482.883,E2 2482.883} C_VEL
LIN {X 0,Y 722.174,Z 783.31,A -85,B 0,C 180,E1 2488.373,E2 2488.373} C_VEL
LIN {X 0,Y 722.325,Z 783.31,A -85,B 0,C 180,E1 2493.872,E2 2493.872} C_VEL
LIN {X 0,Y 722.217,Z 783.31,A -85,B 0,C 180,E1 2499.112,E2 2499.112} C_VEL
LIN {X 0,Y 722.258,Z 783.31,A -85,B 0,C 180,E1 2504.18,E2 2504.18} C_VEL
LIN {X 0,Y 722.41,Z 783.31,A -85,B 0,C 180,E1 2509.125,E2 2509.125} C_VEL
LIN {X 0,Y 722.357,Z 783.31,A -85,B 0,C 180,E1 2513.985,E2 2513.985} C_VEL
LIN {X 0,Y 722.248,Z 783.31,A -85,B 0,C 180,E1 2518.803,E2 2518.803} C_VEL
LIN {X 0,Y 722.248,Z 783.31,A -85,B 0,C 180,E1 2522.409,E2 2522.409} C_VEL
LIN {X 0,Y 722.299,Z 783.31,A -85,B 0,C 180,E1 2526.024,E2 2526.024} C_VEL
LIN {X 0,Y 722.235,Z 783.31,A -85,B 0,C 180,E1 2530.887,E2 2530.887} C_VEL
LIN {X 0,Y 722.298,Z 783.31,A -85,B 0,C 180,E1 2535.828,E2 2535.828} C_VEL
LIN {X 0,Y 722.229,Z 783.31,A -85,B 0,C 180,E1 2540.897,E2 2540.897} C_VEL
LIN {X 0,Y 722.1,Z 783.31,A -85,B 0,C 180,E1 2546.147,E2 2546.147} C_VEL
LIN {X 0,Y 722.078,Z 783.31,A -85,B 0,C 180,E1 2550.65,E2 2550.65} C_VEL
LIN {X 0,Y 722.028,Z 783.31,A -85,B 0,C 180,E1 2555.076,E2 2555.076} C_VEL
LIN {X 0,Y 721.957,Z 783.31,A -85,B 0,C 180,E1 2559.059,E2 2559.059} C_VEL
LIN {X 0,Y 722.203,Z 783.31,A -85,B 0,C 180,E1 2564.497,E2 2564.497} C_VEL
LIN {X 0,Y 721.996,Z 783.31,A -85,B 0,C 180,E1 2569.418,E2 2569.418} C_VEL
LIN {X 0,Y 722.05,Z 783.31,A -85,B 0,C 180,E1 2574.018,E2 2574.018} C_VEL
LIN {X 0,Y 722.19,Z 783.31,A -85,B 0,C 180,E1 2579.337,E2 2579.337} C_VEL
LIN {X 0,Y 722.319,Z 784.04,A -85,B 0,C 180,E1 2581.983,E2 2581.983} C_VEL
LIN {X 0,Y 727.247,Z 796.5,A -85,B 0,C 180,E1 2582.325,E2 2582.325} C_VEL
LIN {X 0,Y 727.095,Z 863.197,A -85,B 0,C 180,E1 2583.154,E2 2583.154} C_VEL
LIN {X 0,Y 726.585,Z 904.849,A -85,B 0,C 180,E1 2584.155,E2 2584.155} C_VEL
LIN {X 0,Y 725.82,Z 944.114,A -85,B 0,C 180,E1 2585.571,E2 2585.571} C_VEL
LIN {X 0,Y 725.009,Z 981.616,A -85,B 0,C 180,E1 2587.424,E2 2587.424} C_VEL
LIN {X 0,Y 724.202,Z 1016.966,A -85,B 0,C 180,E1 2589.727,E2 2589.727} C_VEL
LIN {X 0,Y 723.572,Z 1047.528,A -85,B 0,C 180,E1 2592.299,E2 2592.299} C_VEL
LIN {X 0,Y 723.08,Z 1074.327,A -85,B 0,C 180,E1 2595.206,E2 2595.206} C_VEL
LIN {X 0,Y 722.822,Z 1095.447,A -85,B 0,C 180,E1 2598.208,E2 2598.208} C_VEL
LIN {X 0,Y 722.615,Z 1112.444,A -85,B 0,C 180,E1 2601.561,E2 2601.561} C_VEL
LIN {X 0,Y 722.581,Z 1122.48,A -85,B 0,C 180,E1 2604.568,E2 2604.568} C_VEL
LIN {X 0,Y 722.607,Z 1128.178,A -85,B 0,C 180,E1 2607.598,E2 2607.598} C_VEL
LIN {X 0,Y 722.617,Z 1129.119,A -85,B 0,C 180,E1 2611.202,E2 2611.202} C_VEL
LIN {X 0,Y 722.593,Z 1125.108,A -85,B 0,C 180,E1 2614.21,E2 2614.21} C_VEL
LIN {X 0,Y 722.655,Z 1115.589,A -85,B 0,C 180,E1 2617.531,E2 2617.531} C_VEL
LIN {X 0,Y 722.734,Z 1101.855,A -85,B 0,C 180,E1 2620.58,E2 2620.58} C_VEL
LIN {X 0,Y 722.977,Z 1080.259,A -85,B 0,C 180,E1 2623.947,E2 2623.947} C_VEL
LIN {X 0,Y 723.452,Z 1053.288,A -85,B 0,C 180,E1 2627.051,E2 2627.051} C_VEL
LIN {X 0,Y 724.107,Z 1022.375,A -85,B 0,C 180,E1 2629.773,E2 2629.773} C_VEL
LIN {X 0,Y 724.845,Z 988.216,A -85,B 0,C 180,E1 2632.103,E2 2632.103} C_VEL
LIN {X 0,Y 725.72,Z 949.526,A -85,B 0,C 180,E1 2634.107,E2 2634.107} C_VEL
LIN {X 0,Y 726.489,Z 908.704,A -85,B 0,C 180,E1 2635.644,E2 2635.644} C_VEL
LIN {X 0,Y 727.093,Z 864.587,A -85,B 0,C 180,E1 2636.733,E2 2636.733} C_VEL
LIN {X 0,Y 726.711,Z 794.918,A -85,B 0,C 180,E1 2637.625,E2 2637.625} C_VEL
LIN {X 0,Y 722.423,Z 783.31,A -85,B 0,C 180,E1 2637.96,E2 2637.96} C_VEL
LIN {X 0,Y 722.212,Z 783.31,A -85,B 0,C 180,E1 2643.058,E2 2643.058} C_VEL
LIN {X 0,Y 722.156,Z 783.31,A -85,B 0,C 180,E1 2647.479,E2 2647.479} C_VEL
LIN {X 0,Y 722.166,Z 783.31,A -85,B 0,C 180,E1 2652.749,E2 2652.749} C_VEL
LIN {X 0,Y 721.944,Z 783.31,A -85,B 0,C 180,E1 2657.809,E2 2657.809} C_VEL
LIN {X 0,Y 722.01,Z 783.31,A -85,B 0,C 180,E1 2662.888,E2 2662.888} C_VEL
LIN {X 0,Y 722.142,Z 783.31,A -85,B 0,C 180,E1 2668.361,E2 2668.361} C_VEL
LIN {X 0,Y 722.259,Z 783.31,A -85,B 0,C 180,E1 2673.859,E2 2673.859} C_VEL
LIN {X 0,Y 722.153,Z 783.31,A -85,B 0,C 180,E1 2679.101,E2 2679.101} C_VEL
LIN {X 0,Y 722.253,Z 783.31,A -85,B 0,C 180,E1 2684.171,E2 2684.171} C_VEL
LIN {X 0,Y 722.437,Z 783.31,A -85,B 0,C 180,E1 2689.116,E2 2689.116} C_VEL
LIN {X 0,Y 722.4,Z 783.31,A -85,B 0,C 180,E1 2693.976,E2 2693.976} C_VEL
LIN {X 0,Y 722.286,Z 783.31,A -85,B 0,C 180,E1 2698.794,E2 2698.794} C_VEL
LIN {X 0,Y 722.251,Z 783.31,A -85,B 0,C 180,E1 2702.4,E2 2702.4} C_VEL
LIN {X 0,Y 722.289,Z 783.31,A -85,B 0,C 180,E1 2706.016,E2 2706.016} C_VEL
LIN {X 0,Y 722.275,Z 783.31,A -85,B 0,C 180,E1 2707.809,E2 2707.809} C_VEL
LIN {X 0,Y 719.791,Z 783.31,A -85,B 0,C 180,E1 2708.831,E2 2708.831} C_VEL
LIN {X 0,Y 714.394,Z 783.31,A -85,B 0,C 180,E1 2710.355,E2 2710.355} C_VEL
LIN {X 0,Y 714.3,Z 783.31,A -85,B 0,C 180,E1 2710.532,E2 2710.532} C_VEL
LIN {X 0,Y 714.318,Z 783.31,A -85,B 0,C 180,E1 2714.74,E2 2714.74} C_VEL
LIN {X 0,Y 714.379,Z 783.31,A -85,B 0,C 180,E1 2719.831,E2 2719.831} C_VEL
LIN {X 0,Y 714.279,Z 783.31,A -85,B 0,C 180,E1 2725.096,E2 2725.096} C_VEL
LIN {X 0,Y 714.184,Z 783.31,A -85,B 0,C 180,E1 2729.56,E2 2729.56} C_VEL
LIN {X 0,Y 714.145,Z 783.31,A -85,B 0,C 180,E1 2734.161,E2 2734.161} C_VEL
LIN {X 0,Y 714.11,Z 783.31,A -85,B 0,C 180,E1 2738.273,E2 2738.273} C_VEL
LIN {X 0,Y 714.103,Z 783.31,A -85,B 0,C 180,E1 2742.752,E2 2742.752} C_VEL
LIN {X 0,Y 714.091,Z 783.31,A -85,B 0,C 180,E1 2747.943,E2 2747.943} C_VEL
LIN {X 0,Y 714.309,Z 783.31,A -85,B 0,C 180,E1 2753.696,E2 2753.696} C_VEL
LIN {X 0,Y 714.377,Z 783.31,A -85,B 0,C 180,E1 2758.217,E2 2758.217} C_VEL
LIN {X 0,Y 721.705,Z 802.789,A -85,B 0,C 180,E1 2758.806,E2 2758.806} C_VEL
LIN {X 0,Y 721.351,Z 865.527,A -85,B 0,C 180,E1 2759.646,E2 2759.646} C_VEL
LIN {X 0,Y 720.386,Z 911.012,A -85,B 0,C 180,E1 2760.791,E2 2760.791} C_VEL
LIN {X 0,Y 719.352,Z 953.687,A -85,B 0,C 180,E1 2762.393,E2 2762.393} C_VEL
LIN {X 0,Y 718.285,Z 992.919,A -85,B 0,C 180,E1 2764.377,E2 2764.377} C_VEL
LIN {X 0,Y 717.153,Z 1031,A -85,B 0,C 180,E1 2766.873,E2 2766.873} C_VEL
LIN {X 0,Y 716.233,Z 1064.995,A -85,B 0,C 180,E1 2769.731,E2 2769.731} C_VEL
LIN {X 0,Y 715.417,Z 1094.558,A -85,B 0,C 180,E1 2772.91,E2 2772.91} C_VEL
LIN {X 0,Y 714.952,Z 1118.18,A -85,B 0,C 180,E1 2776.206,E2 2776.206} C_VEL
LIN {X 0,Y 714.797,Z 1135.137,A -85,B 0,C 180,E1 2779.31,E2 2779.31} C_VEL
LIN {X 0,Y 714.659,Z 1148.157,A -85,B 0,C 180,E1 2782.691,E2 2782.691} C_VEL
LIN {X 0,Y 714.657,Z 1155.661,A -85,B 0,C 180,E1 2785.743,E2 2785.743} C_VEL
LIN {X 0,Y 714.625,Z 1159.169,A -85,B 0,C 180,E1 2788.784,E2 2788.784} C_VEL
LIN {X 0,Y 714.729,Z 1158.221,A -85,B 0,C 180,E1 2792.429,E2 2792.429} C_VEL
LIN {X 0,Y 714.683,Z 1151.638,A -85,B 0,C 180,E1 2796.084,E2 2796.084} C_VEL
LIN {X 0,Y 714.762,Z 1140.527,A -85,B 0,C 180,E1 2799.455,E2 2799.455} C_VEL
LIN {X 0,Y 714.965,Z 1122.18,A -85,B 0,C 180,E1 2803.143,E2 2803.143} C_VEL
LIN {X 0,Y 715.318,Z 1099.565,A -85,B 0,C 180,E1 2806.456,E2 2806.456} C_VEL
LIN {X 0,Y 715.947,Z 1073.608,A -85,B 0,C 180,E1 2809.419,E2 2809.419} C_VEL
LIN {X 0,Y 716.894,Z 1040.918,A -85,B 0,C 180,E1 2812.359,E2 2812.359} C_VEL
LIN {X 0,Y 717.996,Z 1004.002,A -85,B 0,C 180,E1 2814.963,E2 2814.963} C_VEL
LIN {X 0,Y 719.222,Z 962.951,A -85,B 0,C 180,E1 2817.185,E2 2817.185} C_VEL
LIN {X 0,Y 720.267,Z 921.647,A -85,B 0,C 180,E1 2818.853,E2 2818.853} C_VEL
LIN {X 0,Y 721.149,Z 880.601,A -85,B 0,C 180,E1 2820.031,E2 2820.031} C_VEL
LIN {X 0,Y 721.61,Z 835.78,A -85,B 0,C 180,E1 2820.816,E2 2820.816} C_VEL
LIN {X 0,Y 720.986,Z 799.019,A -85,B 0,C 180,E1 2821.272,E2 2821.272} C_VEL
LIN {X 0,Y 714.442,Z 783.31,A -85,B 0,C 180,E1 2821.81,E2 2821.81} C_VEL
LIN {X 0,Y 714.273,Z 783.31,A -85,B 0,C 180,E1 2826.437,E2 2826.437} C_VEL
LIN {X 0,Y 714.216,Z 783.31,A -85,B 0,C 180,E1 2832.068,E2 2832.068} C_VEL
LIN {X 0,Y 714.171,Z 783.31,A -85,B 0,C 180,E1 2836.163,E2 2836.163} C_VEL
LIN {X 0,Y 714.1,Z 783.31,A -85,B 0,C 180,E1 2841.724,E2 2841.724} C_VEL
LIN {X 0,Y 714.115,Z 783.31,A -85,B 0,C 180,E1 2846.529,E2 2846.529} C_VEL
LIN {X 0,Y 714.148,Z 783.31,A -85,B 0,C 180,E1 2850.801,E2 2850.801} C_VEL
LIN {X 0,Y 714.307,Z 783.31,A -85,B 0,C 180,E1 2855.795,E2 2855.795} C_VEL
LIN {X 0,Y 714.266,Z 783.31,A -85,B 0,C 180,E1 2860.166,E2 2860.166} C_VEL
LIN {X 0,Y 714.307,Z 783.31,A -85,B 0,C 180,E1 2865.26,E2 2865.26} C_VEL
LIN {X 0,Y 714.437,Z 783.31,A -85,B 0,C 180,E1 2870.237,E2 2870.237} C_VEL
LIN {X 0,Y 714.364,Z 783.31,A -85,B 0,C 180,E1 2875.45,E2 2875.45} C_VEL
LIN {X 0,Y 714.409,Z 783.31,A -85,B 0,C 180,E1 2880.005,E2 2880.005} C_VEL
LIN {X 0,Y 714.607,Z 783.31,A -85,B 0,C 180,E1 2884.869,E2 2884.869} C_VEL
LIN {X 0,Y 714.358,Z 783.31,A -85,B 0,C 180,E1 2889.773,E2 2889.773} C_VEL
LIN {X 0,Y 714.284,Z 783.31,A -85,B 0,C 180,E1 2894.75,E2 2894.75} C_VEL
LIN {X 0,Y 714.31,Z 783.31,A -85,B 0,C 180,E1 2899.842,E2 2899.842} C_VEL
LIN {X 0,Y 714.236,Z 783.31,A -85,B 0,C 180,E1 2905.107,E2 2905.107} C_VEL
LIN {X 0,Y 714.14,Z 783.31,A -85,B 0,C 180,E1 2909.558,E2 2909.558} C_VEL
LIN {X 0,Y 714.125,Z 783.31,A -85,B 0,C 180,E1 2914.163,E2 2914.163} C_VEL
LIN {X 0,Y 714.108,Z 783.31,A -85,B 0,C 180,E1 2918.277,E2 2918.277} C_VEL
LIN {X 0,Y 714.316,Z 783.31,A -85,B 0,C 180,E1 2923.849,E2 2923.849} C_VEL
LIN {X 0,Y 714.049,Z 783.31,A -85,B 0,C 180,E1 2928.869,E2 2928.869} C_VEL
LIN {X 0,Y 714.131,Z 783.31,A -85,B 0,C 180,E1 2933.731,E2 2933.731} C_VEL
LIN {X 0,Y 714.286,Z 783.31,A -85,B 0,C 180,E1 2939.398,E2 2939.398} C_VEL
LIN {X 0,Y 714.342,Z 783.31,A -85,B 0,C 180,E1 2941.626,E2 2941.626} C_VEL
LIN {X 0,Y 720.316,Z 798.849,A -85,B 0,C 180,E1 2942.062,E2 2942.062} C_VEL
LIN {X 0,Y 720.05,Z 864.57,A -85,B 0,C 180,E1 2942.894,E2 2942.894} C_VEL
LIN {X 0,Y 719.422,Z 906.782,A -85,B 0,C 180,E1 2943.937,E2 2943.937} C_VEL
LIN {X 0,Y 718.484,Z 945.989,A -85,B 0,C 180,E1 2945.388,E2 2945.388} C_VEL
LIN {X 0,Y 717.486,Z 983.765,A -85,B 0,C 180,E1 2947.302,E2 2947.302} C_VEL
LIN {X 0,Y 716.586,Z 1018.002,A -85,B 0,C 180,E1 2949.582,E2 2949.582} C_VEL
LIN {X 0,Y 715.817,Z 1049.236,A -85,B 0,C 180,E1 2952.27,E2 2952.27} C_VEL
LIN {X 0,Y 715.292,Z 1074.536,A -85,B 0,C 180,E1 2955.068,E2 2955.068} C_VEL
LIN {X 0,Y 714.986,Z 1095.443,A -85,B 0,C 180,E1 2958.077,E2 2958.077} C_VEL
LIN {X 0,Y 714.757,Z 1112.441,A -85,B 0,C 180,E1 2961.468,E2 2961.468} C_VEL
LIN {X 0,Y 714.693,Z 1122.527,A -85,B 0,C 180,E1 2964.527,E2 2964.527} C_VEL
LIN {X 0,Y 714.701,Z 1128.178,A -85,B 0,C 180,E1 2967.571,E2 2967.571} C_VEL
LIN {X 0,Y 714.715,Z 1129.119,A -85,B 0,C 180,E1 2971.216,E2 2971.216} C_VEL
LIN {X 0,Y 714.603,Z 1124.062,A -85,B 0,C 180,E1 2974.781,E2 2974.781} C_VEL
LIN {X 0,Y 714.686,Z 1113.294,A -85,B 0,C 180,E1 2978.228,E2 2978.228} C_VEL
LIN {X 0,Y 714.851,Z 1098.43,A -85,B 0,C 180,E1 2981.308,E2 2981.308} C_VEL
LIN {X 0,Y 715.176,Z 1077.853,A -85,B 0,C 180,E1 2984.416,E2 2984.416} C_VEL
LIN {X 0,Y 715.728,Z 1052.081,A -85,B 0,C 180,E1 2987.361,E2 2987.361} C_VEL
LIN {X 0,Y 716.51,Z 1020.985,A -85,B 0,C 180,E1 2990.099,E2 2990.099} C_VEL
LIN {X 0,Y 717.423,Z 986.211,A -85,B 0,C 180,E1 2992.464,E2 2992.464} C_VEL
LIN {X 0,Y 718.418,Z 949.542,A -85,B 0,C 180,E1 2994.368,E2 2994.368} C_VEL
LIN {X 0,Y 719.31,Z 908.737,A -85,B 0,C 180,E1 2995.919,E2 2995.919} C_VEL
LIN {X 0,Y 720.003,Z 865.653,A -85,B 0,C 180,E1 2996.998,E2 2996.998} C_VEL
LIN {X 0,Y 719.916,Z 797.679,A -85,B 0,C 180,E1 2997.878,E2 2997.878} C_VEL
LIN {X 0,Y 714.448,Z 783.31,A -85,B 0,C 180,E1 2998.325,E2 2998.325} C_VEL
LIN {X 0,Y 714.22,Z 783.31,A -85,B 0,C 180,E1 3003.476,E2 3003.476} C_VEL
LIN {X 0,Y 714.118,Z 783.31,A -85,B 0,C 180,E1 3008.275,E2 3008.275} C_VEL
LIN {X 0,Y 714.328,Z 783.31,A -85,B 0,C 180,E1 3013.847,E2 3013.847} C_VEL
LIN {X 0,Y 714.051,Z 783.31,A -85,B 0,C 180,E1 3018.867,E2 3018.867} C_VEL
LIN {X 0,Y 714.121,Z 783.31,A -85,B 0,C 180,E1 3023.733,E2 3023.733} C_VEL
LIN {X 0,Y 714.241,Z 783.31,A -85,B 0,C 180,E1 3029.392,E2 3029.392} C_VEL
LIN {X 0,Y 714.299,Z 783.31,A -85,B 0,C 180,E1 3034.895,E2 3034.895} C_VEL
LIN {X 0,Y 714.279,Z 783.31,A -85,B 0,C 180,E1 3038.966,E2 3038.966} C_VEL
LIN {X 0,Y 714.34,Z 783.31,A -85,B 0,C 180,E1 3043.991,E2 3043.991} C_VEL
LIN {X 0,Y 714.491,Z 783.31,A -85,B 0,C 180,E1 3048.994,E2 3048.994} C_VEL
LIN {X 0,Y 714.508,Z 783.31,A -85,B 0,C 180,E1 3053.91,E2 3053.91} C_VEL
LIN {X 0,Y 714.386,Z 783.31,A -85,B 0,C 180,E1 3058.78,E2 3058.78} C_VEL
LIN {X 0,Y 714.35,Z 783.31,A -85,B 0,C 180,E1 3062.426,E2 3062.426} C_VEL
LIN {X 0,Y 714.379,Z 783.31,A -85,B 0,C 180,E1 3066.082,E2 3066.082} C_VEL
LIN {X 0,Y 714.3,Z 783.31,A -85,B 0,C 180,E1 3070.532,E2 3070.532} C_VEL
LIN {X 0,Y 710.37,Z 783.31,A -85,B 0,C 180,E1 3071.905,E2 3071.905} C_VEL
LIN {X 0,Y 706.436,Z 783.31,A -85,B 0,C 180,E1 3073.294,E2 3073.294} C_VEL
LIN {X 0,Y 706.496,Z 783.31,A -85,B 0,C 180,E1 3077.466,E2 3077.466} C_VEL
LIN {X 0,Y 706.353,Z 783.31,A -85,B 0,C 180,E1 3082.722,E2 3082.722} C_VEL
LIN {X 0,Y 706.309,Z 783.31,A -85,B 0,C 180,E1 3088.152,E2 3088.152} C_VEL
LIN {X 0,Y 706.28,Z 783.31,A -85,B 0,C 180,E1 3093.21,E2 3093.21} C_VEL
LIN {X 0,Y 706.175,Z 783.31,A -85,B 0,C 180,E1 3098.468,E2 3098.468} C_VEL
LIN {X 0,Y 706.159,Z 783.31,A -85,B 0,C 180,E1 3103.351,E2 3103.351} C_VEL
LIN {X 0,Y 706.152,Z 783.31,A -85,B 0,C 180,E1 3108.662,E2 3108.662} C_VEL
LIN {X 0,Y 706.321,Z 783.31,A -85,B 0,C 180,E1 3113.083,E2 3113.083} C_VEL
LIN {X 0,Y 706.465,Z 784.095,A -85,B 0,C 180,E1 3117.835,E2 3117.835} C_VEL
LIN {X 0,Y 714.941,Z 803.665,A -85,B 0,C 180,E1 3118.487,E2 3118.487} C_VEL
LIN {X 0,Y 714.517,Z 865.526,A -85,B 0,C 180,E1 3119.324,E2 3119.324} C_VEL
LIN {X 0,Y 713.383,Z 911.365,A -85,B 0,C 180,E1 3120.487,E2 3120.487} C_VEL
LIN {X 0,Y 712.23,Z 953.692,A -85,B 0,C 180,E1 3122.093,E2 3122.093} C_VEL
LIN {X 0,Y 710.983,Z 992.915,A -85,B 0,C 180,E1 3124.094,E2 3124.094} C_VEL
LIN {X 0,Y 709.731,Z 1030.896,A -85,B 0,C 180,E1 3126.609,E2 3126.609} C_VEL
LIN {X 0,Y 708.615,Z 1064.994,A -85,B 0,C 180,E1 3129.504,E2 3129.504} C_VEL
LIN {X 0,Y 707.695,Z 1094.556,A -85,B 0,C 180,E1 3132.718,E2 3132.718} C_VEL
LIN {X 0,Y 707.131,Z 1118.181,A -85,B 0,C 180,E1 3136.05,E2 3136.05} C_VEL
LIN {X 0,Y 706.96,Z 1135.138,A -85,B 0,C 180,E1 3139.19,E2 3139.19} C_VEL
LIN {X 0,Y 706.773,Z 1148.157,A -85,B 0,C 180,E1 3142.609,E2 3142.609} C_VEL
LIN {X 0,Y 706.751,Z 1155.813,A -85,B 0,C 180,E1 3145.774,E2 3145.774} C_VEL
LIN {X 0,Y 706.736,Z 1159.169,A -85,B 0,C 180,E1 3148.77,E2 3148.77} C_VEL
LIN {X 0,Y 706.823,Z 1158.22,A -85,B 0,C 180,E1 3152.456,E2 3152.456} C_VEL
LIN {X 0,Y 706.775,Z 1151.639,A -85,B 0,C 180,E1 3156.152,E2 3156.152} C_VEL
LIN {X 0,Y 706.875,Z 1140.104,A -85,B 0,C 180,E1 3159.659,E2 3159.659} C_VEL
LIN {X 0,Y 707.098,Z 1121.871,A -85,B 0,C 180,E1 3163.347,E2 3163.347} C_VEL
LIN {X 0,Y 707.544,Z 1099.566,A -85,B 0,C 180,E1 3166.642,E2 3166.642} C_VEL
LIN {X 0,Y 708.308,Z 1072.281,A -85,B 0,C 180,E1 3169.771,E2 3169.771} C_VEL
LIN {X 0,Y 709.354,Z 1040.919,A -85,B 0,C 180,E1 3172.61,E2 3172.61} C_VEL
LIN {X 0,Y 710.657,Z 1004.003,A -85,B 0,C 180,E1 3175.239,E2 3175.239} C_VEL
LIN {X 0,Y 712.027,Z 962.955,A -85,B 0,C 180,E1 3177.482,E2 3177.482} C_VEL
LIN {X 0,Y 713.279,Z 921.76,A -85,B 0,C 180,E1 3179.158,E2 3179.158} C_VEL
LIN {X 0,Y 714.289,Z 880.862,A -85,B 0,C 180,E1 3180.344,E2 3180.344} C_VEL
LIN {X 0,Y 714.82,Z 836.097,A -85,B 0,C 180,E1 3181.137,E2 3181.137} C_VEL
LIN {X 0,Y 714.449,Z 801.898,A -85,B 0,C 180,E1 3181.558,E2 3181.558} C_VEL
LIN {X 0,Y 706.469,Z 783.31,A -85,B 0,C 180,E1 3182.245,E2 3182.245} C_VEL
LIN {X 0,Y 706.279,Z 783.31,A -85,B 0,C 180,E1 3187.477,E2 3187.477} C_VEL
LIN {X 0,Y 706.416,Z 783.31,A -85,B 0,C 180,E1 3193.341,E2 3193.341} C_VEL
LIN {X 0,Y 706.171,Z 783.31,A -85,B 0,C 180,E1 3198.672,E2 3198.672} C_VEL
LIN {X 0,Y 706.169,Z 783.31,A -85,B 0,C 180,E1 3203.085,E2 3203.085} C_VEL
LIN {X 0,Y 706.238,Z 783.31,A -85,B 0,C 180,E1 3207.573,E2 3207.573} C_VEL
LIN {X 0,Y 706.42,Z 783.31,A -85,B 0,C 180,E1 3213.237,E2 3213.237} C_VEL
LIN {X 0,Y 706.405,Z 783.31,A -85,B 0,C 180,E1 3218.622,E2 3218.622} C_VEL
LIN {X 0,Y 706.435,Z 783.31,A -85,B 0,C 180,E1 3223.816,E2 3223.816} C_VEL
LIN {X 0,Y 706.519,Z 783.31,A -85,B 0,C 180,E1 3228.877,E2 3228.877} C_VEL
LIN {X 0,Y 706.555,Z 783.31,A -85,B 0,C 180,E1 3233.85,E2 3233.85} C_VEL
LIN {X 0,Y 706.45,Z 783.31,A -85,B 0,C 180,E1 3238.776,E2 3238.776} C_VEL
LIN {X 0,Y 706.463,Z 783.31,A -85,B 0,C 180,E1 3242.463,E2 3242.463} C_VEL
LIN {X 0,Y 706.498,Z 783.31,A -85,B 0,C 180,E1 3246.16,E2 3246.16} C_VEL
LIN {X 0,Y 706.423,Z 783.31,A -85,B 0,C 180,E1 3251.134,E2 3251.134} C_VEL
LIN {X 0,Y 706.455,Z 783.31,A -85,B 0,C 180,E1 3256.193,E2 3256.193} C_VEL
LIN {X 0,Y 706.341,Z 783.31,A -85,B 0,C 180,E1 3261.39,E2 3261.39} C_VEL
LIN {X 0,Y 706.277,Z 783.31,A -85,B 0,C 180,E1 3265.71,E2 3265.71} C_VEL
LIN {X 0,Y 706.28,Z 783.31,A -85,B 0,C 180,E1 3270.991,E2 3270.991} C_VEL
LIN {X 0,Y 706.237,Z 783.31,A -85,B 0,C 180,E1 3275.4,E2 3275.4} C_VEL
LIN {X 0,Y 706.078,Z 783.31,A -85,B 0,C 180,E1 3280.075,E2 3280.075} C_VEL
LIN {X 0,Y 706.329,Z 783.31,A -85,B 0,C 180,E1 3285.065,E2 3285.065} C_VEL
LIN {X 0,Y 706.176,Z 783.31,A -85,B 0,C 180,E1 3290.572,E2 3290.572} C_VEL
LIN {X 0,Y 706.204,Z 783.31,A -85,B 0,C 180,E1 3296.095,E2 3296.095} C_VEL
LIN {X 0,Y 706.379,Z 783.31,A -85,B 0,C 180,E1 3301.284,E2 3301.284} C_VEL
LIN {X 0,Y 713.254,Z 800.855,A -85,B 0,C 180,E1 3301.784,E2 3301.784} C_VEL
LIN {X 0,Y 713.003,Z 864.638,A -85,B 0,C 180,E1 3302.605,E2 3302.605} C_VEL
LIN {X 0,Y 712.245,Z 907.603,A -85,B 0,C 180,E1 3303.68,E2 3303.68} C_VEL
LIN {X 0,Y 711.11,Z 948.74,A -85,B 0,C 180,E1 3305.238,E2 3305.238} C_VEL
LIN {X 0,Y 709.965,Z 987.902,A -85,B 0,C 180,E1 3307.298,E2 3307.298} C_VEL
LIN {X 0,Y 708.821,Z 1024.268,A -85,B 0,C 180,E1 3309.839,E2 3309.839} C_VEL
LIN {X 0,Y 707.894,Z 1055.731,A -85,B 0,C 180,E1 3312.725,E2 3312.725} C_VEL
LIN {X 0,Y 707.296,Z 1080.952,A -85,B 0,C 180,E1 3315.739,E2 3315.739} C_VEL
LIN {X 0,Y 706.968,Z 1100.691,A -85,B 0,C 180,E1 3318.88,E2 3318.88} C_VEL
LIN {X 0,Y 706.815,Z 1114.786,A -85,B 0,C 180,E1 3321.992,E2 3321.992} C_VEL
LIN {X 0,Y 706.754,Z 1124.076,A -85,B 0,C 180,E1 3325.082,E2 3325.082} C_VEL
LIN {X 0,Y 706.796,Z 1128.177,A -85,B 0,C 180,E1 3327.544,E2 3327.544} C_VEL
LIN {X 0,Y 706.827,Z 1129.12,A -85,B 0,C 180,E1 3331.229,E2 3331.229} C_VEL
LIN {X 0,Y 706.798,Z 1125.417,A -85,B 0,C 180,E1 3334.147,E2 3334.147} C_VEL
LIN {X 0,Y 706.891,Z 1116.741,A -85,B 0,C 180,E1 3337.39,E2 3337.39} C_VEL
LIN {X 0,Y 707,Z 1101.908,A -85,B 0,C 180,E1 3340.809,E2 3340.809} C_VEL
LIN {X 0,Y 707.316,Z 1080.264,A -85,B 0,C 180,E1 3344.262,E2 3344.262} C_VEL
LIN {X 0,Y 707.979,Z 1054.883,A -85,B 0,C 180,E1 3347.275,E2 3347.275} C_VEL
LIN {X 0,Y 708.876,Z 1023.084,A -85,B 0,C 180,E1 3350.162,E2 3350.162} C_VEL
LIN {X 0,Y 709.94,Z 988.24,A -85,B 0,C 180,E1 3352.593,E2 3352.593} C_VEL
LIN {X 0,Y 711.13,Z 949.516,A -85,B 0,C 180,E1 3354.636,E2 3354.636} C_VEL
LIN {X 0,Y 712.162,Z 908.747,A -85,B 0,C 180,E1 3356.199,E2 3356.199} C_VEL
LIN {X 0,Y 712.998,Z 864.815,A -85,B 0,C 180,E1 3357.302,E2 3357.302} C_VEL
LIN {X 0,Y 712.592,Z 798.887,A -85,B 0,C 180,E1 3358.177,E2 3358.177} C_VEL
LIN {X 0,Y 706.483,Z 783.31,A -85,B 0,C 180,E1 3358.624,E2 3358.624} C_VEL
LIN {X 0,Y 706.278,Z 783.31,A -85,B 0,C 180,E1 3363.903,E2 3363.903} C_VEL
LIN {X 0,Y 706.185,Z 783.31,A -85,B 0,C 180,E1 3368.479,E2 3368.479} C_VEL
LIN {X 0,Y 706.37,Z 783.31,A -85,B 0,C 180,E1 3373.347,E2 3373.347} C_VEL
LIN {X 0,Y 706.163,Z 783.31,A -85,B 0,C 180,E1 3378.676,E2 3378.676} C_VEL
LIN {X 0,Y 706.123,Z 783.31,A -85,B 0,C 180,E1 3383.07,E2 3383.07} C_VEL
LIN {X 0,Y 706.208,Z 783.31,A -85,B 0,C 180,E1 3387.561,E2 3387.561} C_VEL
LIN {X 0,Y 706.26,Z 783.31,A -85,B 0,C 180,E1 3391.835,E2 3391.835} C_VEL
LIN {X 0,Y 706.378,Z 783.31,A -85,B 0,C 180,E1 3395.947,E2 3395.947} C_VEL
LIN {X 0,Y 706.395,Z 783.31,A -85,B 0,C 180,E1 3401.229,E2 3401.229} C_VEL
LIN {X 0,Y 706.343,Z 783.31,A -85,B 0,C 180,E1 3406.348,E2 3406.348} C_VEL
LIN {X 0,Y 706.52,Z 783.31,A -85,B 0,C 180,E1 3410.577,E2 3410.577} C_VEL
LIN {X 0,Y 706.474,Z 783.31,A -85,B 0,C 180,E1 3415.075,E2 3415.075} C_VEL
LIN {X 0,Y 706.547,Z 783.31,A -85,B 0,C 180,E1 3419.995,E2 3419.995} C_VEL
LIN {X 0,Y 706.67,Z 783.31,A -85,B 0,C 180,E1 3424.915,E2 3424.915} C_VEL
LIN {X 0,Y 706.471,Z 783.31,A -85,B 0,C 180,E1 3429.874,E2 3429.874} C_VEL
LIN {X 0,Y 706.436,Z 783.31,A -85,B 0,C 180,E1 3433.294,E2 3433.294} C_VEL
LIN {X 0,Y 705.179,Z 783.31,A -85,B 0,C 180,E1 3433.998,E2 3433.998} C_VEL
LIN {X 0,Y 698.631,Z 783.31,A -85,B 0,C 180,E1 3435.907,E2 3435.907} C_VEL
LIN {X 0,Y 698.56,Z 783.31,A -85,B 0,C 180,E1 3436.088,E2 3436.088} C_VEL
LIN {X 0,Y 698.48,Z 783.31,A -85,B 0,C 180,E1 3441.127,E2 3441.127} C_VEL
LIN {X 0,Y 698.438,Z 783.31,A -85,B 0,C 180,E1 3445.706,E2 3445.706} C_VEL
LIN {X 0,Y 698.375,Z 783.31,A -85,B 0,C 180,E1 3449.925,E2 3449.925} C_VEL
LIN {X 0,Y 698.298,Z 783.31,A -85,B 0,C 180,E1 3454.458,E2 3454.458} C_VEL
LIN {X 0,Y 698.225,Z 783.31,A -85,B 0,C 180,E1 3458.989,E2 3458.989} C_VEL
LIN {X 0,Y 698.161,Z 783.31,A -85,B 0,C 180,E1 3464.259,E2 3464.259} C_VEL
LIN {X 0,Y 698.176,Z 783.31,A -85,B 0,C 180,E1 3469.412,E2 3469.412} C_VEL
LIN {X 0,Y 698.397,Z 783.31,A -85,B 0,C 180,E1 3474.142,E2 3474.142} C_VEL
LIN {X 0,Y 698.448,Z 783.31,A -85,B 0,C 180,E1 3477.399,E2 3477.399} C_VEL
LIN {X 0,Y 708.177,Z 805.417,A -85,B 0,C 180,E1 3478.171,E2 3478.171} C_VEL
LIN {X 0,Y 707.697,Z 865.812,A -85,B 0,C 180,E1 3479.002,E2 3479.002} C_VEL
LIN {X 0,Y 706.442,Z 910.973,A -85,B 0,C 180,E1 3480.155,E2 3480.155} C_VEL
LIN {X 0,Y 705.155,Z 953.692,A -85,B 0,C 180,E1 3481.788,E2 3481.788} C_VEL
LIN {X 0,Y 703.648,Z 994.143,A -85,B 0,C 180,E1 3483.88,E2 3483.88} C_VEL
LIN {X 0,Y 702.253,Z 1030.894,A -85,B 0,C 180,E1 3486.345,E2 3486.345} C_VEL
LIN {X 0,Y 700.993,Z 1064.992,A -85,B 0,C 180,E1 3489.271,E2 3489.271} C_VEL
LIN {X 0,Y 699.926,Z 1095.881,A -85,B 0,C 180,E1 3492.682,E2 3492.682} C_VEL
LIN {X 0,Y 699.266,Z 1120.136,A -85,B 0,C 180,E1 3496.21,E2 3496.21} C_VEL
LIN {X 0,Y 698.989,Z 1137.835,A -85,B 0,C 180,E1 3499.697,E2 3499.697} C_VEL
LIN {X 0,Y 698.862,Z 1150.067,A -85,B 0,C 180,E1 3503.151,E2 3503.151} C_VEL
LIN {X 0,Y 698.777,Z 1156.651,A -85,B 0,C 180,E1 3506.269,E2 3506.269} C_VEL
LIN {X 0,Y 698.8,Z 1159.5,A -85,B 0,C 180,E1 3509.999,E2 3509.999} C_VEL
LIN {X 0,Y 698.828,Z 1156.654,A -85,B 0,C 180,E1 3513.728,E2 3513.728} C_VEL
LIN {X 0,Y 698.839,Z 1150.073,A -85,B 0,C 180,E1 3516.848,E2 3516.848} C_VEL
LIN {X 0,Y 698.922,Z 1137.845,A -85,B 0,C 180,E1 3520.302,E2 3520.302} C_VEL
LIN {X 0,Y 699.275,Z 1121.727,A -85,B 0,C 180,E1 3523.526,E2 3523.526} C_VEL
LIN {X 0,Y 699.775,Z 1098.353,A -85,B 0,C 180,E1 3526.995,E2 3526.995} C_VEL
LIN {X 0,Y 700.668,Z 1071.086,A -85,B 0,C 180,E1 3530.119,E2 3530.119} C_VEL
LIN {X 0,Y 701.929,Z 1038.881,A -85,B 0,C 180,E1 3533.026,E2 3533.026} C_VEL
LIN {X 0,Y 703.407,Z 1001.574,A -85,B 0,C 180,E1 3535.669,E2 3535.669} C_VEL
LIN {X 0,Y 704.997,Z 960.05,A -85,B 0,C 180,E1 3537.924,E2 3537.924} C_VEL
LIN {X 0,Y 706.406,Z 917.664,A -85,B 0,C 180,E1 3539.618,E2 3539.618} C_VEL
LIN {X 0,Y 707.509,Z 877.208,A -85,B 0,C 180,E1 3540.749,E2 3540.749} C_VEL
LIN {X 0,Y 708.082,Z 833.227,A -85,B 0,C 180,E1 3541.507,E2 3541.507} C_VEL
LIN {X 0,Y 707.534,Z 803.969,A -85,B 0,C 180,E1 3541.878,E2 3541.878} C_VEL
LIN {X 0,Y 698.5,Z 783.31,A -85,B 0,C 180,E1 3542.629,E2 3542.629} C_VEL
LIN {X 0,Y 698.398,Z 783.31,A -85,B 0,C 180,E1 3547.404,E2 3547.404} C_VEL
LIN {X 0,Y 698.378,Z 783.31,A -85,B 0,C 180,E1 3552.481,E2 3552.481} C_VEL
LIN {X 0,Y 698.21,Z 783.31,A -85,B 0,C 180,E1 3557.734,E2 3557.734} C_VEL
LIN {X 0,Y 698.278,Z 783.31,A -85,B 0,C 180,E1 3562.597,E2 3562.597} C_VEL
LIN {X 0,Y 698.32,Z 783.31,A -85,B 0,C 180,E1 3567.798,E2 3567.798} C_VEL
LIN {X 0,Y 698.448,Z 783.31,A -85,B 0,C 180,E1 3572.907,E2 3572.907} C_VEL
LIN {X 0,Y 698.556,Z 783.31,A -85,B 0,C 180,E1 3577.027,E2 3577.027} C_VEL
LIN {X 0,Y 698.566,Z 783.31,A -85,B 0,C 180,E1 3582.616,E2 3582.616} C_VEL
LIN {X 0,Y 698.395,Z 783.31,A -85,B 0,C 180,E1 3587.488,E2 3587.488} C_VEL
LIN {X 0,Y 698.617,Z 783.31,A -85,B 0,C 180,E1 3592.528,E2 3592.528} C_VEL
LIN {X 0,Y 698.713,Z 783.31,A -85,B 0,C 180,E1 3597.519,E2 3597.519} C_VEL
LIN {X 0,Y 698.562,Z 783.31,A -85,B 0,C 180,E1 3602.491,E2 3602.491} C_VEL
LIN {X 0,Y 698.599,Z 783.31,A -85,B 0,C 180,E1 3606.23,E2 3606.23} C_VEL
LIN {X 0,Y 698.516,Z 783.31,A -85,B 0,C 180,E1 3611.261,E2 3611.261} C_VEL
LIN {X 0,Y 698.528,Z 783.31,A -85,B 0,C 180,E1 3616.382,E2 3616.382} C_VEL
LIN {X 0,Y 698.422,Z 783.31,A -85,B 0,C 180,E1 3621.644,E2 3621.644} C_VEL
LIN {X 0,Y 698.397,Z 783.31,A -85,B 0,C 180,E1 3625.718,E2 3625.718} C_VEL
LIN {X 0,Y 698.324,Z 783.31,A -85,B 0,C 180,E1 3629.938,E2 3629.938} C_VEL
LIN {X 0,Y 698.273,Z 783.31,A -85,B 0,C 180,E1 3634.459,E2 3634.459} C_VEL
LIN {X 0,Y 698.23,Z 783.31,A -85,B 0,C 180,E1 3639,E2 3639} C_VEL
LIN {X 0,Y 698.381,Z 783.31,A -85,B 0,C 180,E1 3644.281,E2 3644.281} C_VEL
LIN {X 0,Y 698.234,Z 783.31,A -85,B 0,C 180,E1 3649.421,E2 3649.421} C_VEL
LIN {X 0,Y 698.236,Z 783.31,A -85,B 0,C 180,E1 3654.135,E2 3654.135} C_VEL
LIN {X 0,Y 698.374,Z 783.31,A -85,B 0,C 180,E1 3658.623,E2 3658.623} C_VEL
LIN {X 0,Y 698.476,Z 783.486,A -85,B 0,C 180,E1 3660.932,E2 3660.932} C_VEL
LIN {X 0,Y 706.399,Z 805.09,A -85,B 0,C 180,E1 3661.533,E2 3661.533} C_VEL
LIN {X 0,Y 705.96,Z 865.739,A -85,B 0,C 180,E1 3662.331,E2 3662.331} C_VEL
LIN {X 0,Y 705.085,Z 909.031,A -85,B 0,C 180,E1 3663.436,E2 3663.436} C_VEL
LIN {X 0,Y 703.786,Z 950.741,A -85,B 0,C 180,E1 3665.054,E2 3665.054} C_VEL
LIN {X 0,Y 702.48,Z 989.762,A -85,B 0,C 180,E1 3667.156,E2 3667.156} C_VEL
LIN {X 0,Y 701.233,Z 1024.262,A -85,B 0,C 180,E1 3669.611,E2 3669.611} C_VEL
LIN {X 0,Y 700.188,Z 1055.727,A -85,B 0,C 180,E1 3672.529,E2 3672.529} C_VEL
LIN {X 0,Y 699.508,Z 1080.949,A -85,B 0,C 180,E1 3675.577,E2 3675.577} C_VEL
LIN {X 0,Y 699.11,Z 1100.688,A -85,B 0,C 180,E1 3678.753,E2 3678.753} C_VEL
LIN {X 0,Y 698.952,Z 1114.784,A -85,B 0,C 180,E1 3681.901,E2 3681.901} C_VEL
LIN {X 0,Y 698.88,Z 1124.074,A -85,B 0,C 180,E1 3685.026,E2 3685.026} C_VEL
LIN {X 0,Y 698.891,Z 1128.176,A -85,B 0,C 180,E1 3687.516,E2 3687.516} C_VEL
LIN {X 0,Y 698.925,Z 1129.12,A -85,B 0,C 180,E1 3691.243,E2 3691.243} C_VEL
LIN {X 0,Y 698.901,Z 1125.284,A -85,B 0,C 180,E1 3694.264,E2 3694.264} C_VEL
LIN {X 0,Y 698.991,Z 1116.744,A -85,B 0,C 180,E1 3697.474,E2 3697.474} C_VEL
LIN {X 0,Y 699.135,Z 1101.91,A -85,B 0,C 180,E1 3700.932,E2 3700.932} C_VEL
LIN {X 0,Y 699.52,Z 1080.267,A -85,B 0,C 180,E1 3704.425,E2 3704.425} C_VEL
LIN {X 0,Y 700.227,Z 1054.889,A -85,B 0,C 180,E1 3707.472,E2 3707.472} C_VEL
LIN {X 0,Y 701.287,Z 1023.092,A -85,B 0,C 180,E1 3710.39,E2 3710.39} C_VEL
LIN {X 0,Y 702.493,Z 988.253,A -85,B 0,C 180,E1 3712.846,E2 3712.846} C_VEL
LIN {X 0,Y 703.859,Z 949.3,A -85,B 0,C 180,E1 3714.918,E2 3714.918} C_VEL
LIN {X 0,Y 705.051,Z 908.768,A -85,B 0,C 180,E1 3716.483,E2 3716.483} C_VEL
LIN {X 0,Y 705.93,Z 866.137,A -85,B 0,C 180,E1 3717.572,E2 3717.572} C_VEL
LIN {X 0,Y 705.917,Z 801.78,A -85,B 0,C 180,E1 3718.435,E2 3718.435} C_VEL
LIN {X 0,Y 698.531,Z 783.31,A -85,B 0,C 180,E1 3719.032,E2 3719.032} C_VEL
LIN {X 0,Y 698.32,Z 783.31,A -85,B 0,C 180,E1 3724.462,E2 3724.462} C_VEL
LIN {X 0,Y 698.242,Z 783.31,A -85,B 0,C 180,E1 3728.999,E2 3728.999} C_VEL
LIN {X 0,Y 698.393,Z 783.31,A -85,B 0,C 180,E1 3734.279,E2 3734.279} C_VEL
LIN {X 0,Y 698.217,Z 783.31,A -85,B 0,C 180,E1 3739.423,E2 3739.423} C_VEL
LIN {X 0,Y 698.242,Z 783.31,A -85,B 0,C 180,E1 3744.132,E2 3744.132} C_VEL
LIN {X 0,Y 698.334,Z 783.31,A -85,B 0,C 180,E1 3748.617,E2 3748.617} C_VEL
LIN {X 0,Y 698.417,Z 783.31,A -85,B 0,C 180,E1 3752.895,E2 3752.895} C_VEL
LIN {X 0,Y 698.518,Z 783.31,A -85,B 0,C 180,E1 3757.015,E2 3757.015} C_VEL
LIN {X 0,Y 698.56,Z 783.31,A -85,B 0,C 180,E1 3762.625,E2 3762.625} C_VEL
LIN {X 0,Y 698.443,Z 783.31,A -85,B 0,C 180,E1 3767.48,E2 3767.48} C_VEL
LIN {X 0,Y 698.706,Z 783.31,A -85,B 0,C 180,E1 3772.52,E2 3772.52} C_VEL
LIN {X 0,Y 698.703,Z 783.31,A -85,B 0,C 180,E1 3777.51,E2 3777.51} C_VEL
LIN {X 0,Y 698.564,Z 783.31,A -85,B 0,C 180,E1 3782.481,E2 3782.481} C_VEL
LIN {X 0,Y 698.576,Z 783.31,A -85,B 0,C 180,E1 3786.221,E2 3786.221} C_VEL
LIN {X 0,Y 698.515,Z 783.31,A -85,B 0,C 180,E1 3791.252,E2 3791.252} C_VEL
LIN {X 0,Y 698.56,Z 783.31,A -85,B 0,C 180,E1 3796.088,E2 3796.088} C_VEL
LIN {X 0,Y 696.067,Z 783.31,A -85,B 0,C 180,E1 3797.148,E2 3797.148} C_VEL
LIN {X 0,Y 690.664,Z 783.31,A -85,B 0,C 180,E1 3798.73,E2 3798.73} C_VEL
LIN {X 0,Y 690.577,Z 783.31,A -85,B 0,C 180,E1 3798.913,E2 3798.913} C_VEL
LIN {X 0,Y 690.53,Z 783.31,A -85,B 0,C 180,E1 3803.256,E2 3803.256} C_VEL
LIN {X 0,Y 690.497,Z 783.31,A -85,B 0,C 180,E1 3808.629,E2 3808.629} C_VEL
LIN {X 0,Y 690.396,Z 783.31,A -85,B 0,C 180,E1 3813.491,E2 3813.491} C_VEL
LIN {X 0,Y 690.377,Z 783.31,A -85,B 0,C 180,E1 3817.906,E2 3817.906} C_VEL
LIN {X 0,Y 690.247,Z 783.31,A -85,B 0,C 180,E1 3823.581,E2 3823.581} C_VEL
LIN {X 0,Y 690.223,Z 783.31,A -85,B 0,C 180,E1 3828.809,E2 3828.809} C_VEL
LIN {X 0,Y 690.5,Z 783.31,A -85,B 0,C 180,E1 3834.266,E2 3834.266} C_VEL
LIN {X 0,Y 690.55,Z 783.887,A -85,B 0,C 180,E1 3836.998,E2 3836.998} C_VEL
LIN {X 0,Y 701.541,Z 808.697,A -85,B 0,C 180,E1 3837.873,E2 3837.873} C_VEL
LIN {X 0,Y 700.937,Z 865.811,A -85,B 0,C 180,E1 3838.67,E2 3838.67} C_VEL
LIN {X 0,Y 699.51,Z 911.924,A -85,B 0,C 180,E1 3839.859,E2 3839.859} C_VEL
LIN {X 0,Y 698.011,Z 955.057,A -85,B 0,C 180,E1 3841.537,E2 3841.537} C_VEL
LIN {X 0,Y 696.378,Z 994.528,A -85,B 0,C 180,E1 3843.611,E2 3843.611} C_VEL
LIN {X 0,Y 694.771,Z 1031.487,A -85,B 0,C 180,E1 3846.123,E2 3846.123} C_VEL
LIN {X 0,Y 693.304,Z 1066.646,A -85,B 0,C 180,E1 3849.197,E2 3849.197} C_VEL
LIN {X 0,Y 692.175,Z 1095.88,A -85,B 0,C 180,E1 3852.482,E2 3852.482} C_VEL
LIN {X 0,Y 691.451,Z 1120.135,A -85,B 0,C 180,E1 3856.051,E2 3856.051} C_VEL
LIN {X 0,Y 691.134,Z 1137.835,A -85,B 0,C 180,E1 3859.579,E2 3859.579} C_VEL
LIN {X 0,Y 690.987,Z 1150.067,A -85,B 0,C 180,E1 3863.072,E2 3863.072} C_VEL
LIN {X 0,Y 690.895,Z 1156.65,A -85,B 0,C 180,E1 3866.227,E2 3866.227} C_VEL
LIN {X 0,Y 690.902,Z 1159.5,A -85,B 0,C 180,E1 3869.999,E2 3869.999} C_VEL
LIN {X 0,Y 690.94,Z 1156.654,A -85,B 0,C 180,E1 3873.771,E2 3873.771} C_VEL
LIN {X 0,Y 690.958,Z 1150.073,A -85,B 0,C 180,E1 3876.926,E2 3876.926} C_VEL
LIN {X 0,Y 691.062,Z 1137.845,A -85,B 0,C 180,E1 3880.42,E2 3880.42} C_VEL
LIN {X 0,Y 691.421,Z 1121.558,A -85,B 0,C 180,E1 3883.712,E2 3883.712} C_VEL
LIN {X 0,Y 692.05,Z 1098.354,A -85,B 0,C 180,E1 3887.19,E2 3887.19} C_VEL
LIN {X 0,Y 693.033,Z 1071.508,A -85,B 0,C 180,E1 3890.306,E2 3890.306} C_VEL
LIN {X 0,Y 694.393,Z 1039.687,A -85,B 0,C 180,E1 3893.225,E2 3893.225} C_VEL
LIN {X 0,Y 696.037,Z 1002.847,A -85,B 0,C 180,E1 3895.881,E2 3895.881} C_VEL
LIN {X 0,Y 697.845,Z 961.462,A -85,B 0,C 180,E1 3898.166,E2 3898.166} C_VEL
LIN {X 0,Y 699.42,Z 919.32,A -85,B 0,C 180,E1 3899.883,E2 3899.883} C_VEL
LIN {X 0,Y 700.684,Z 879.511,A -85,B 0,C 180,E1 3901.028,E2 3901.028} C_VEL
LIN {X 0,Y 701.351,Z 834.673,A -85,B 0,C 180,E1 3901.824,E2 3901.824} C_VEL
LIN {X 0,Y 700.88,Z 806.545,A -85,B 0,C 180,E1 3902.186,E2 3902.186} C_VEL
LIN {X 0,Y 690.521,Z 783.31,A -85,B 0,C 180,E1 3903.087,E2 3903.087} C_VEL
LIN {X 0,Y 690.455,Z 783.31,A -85,B 0,C 180,E1 3907.91,E2 3907.91} C_VEL
LIN {X 0,Y 690.486,Z 783.31,A -85,B 0,C 180,E1 3913.616,E2 3913.616} C_VEL
LIN {X 0,Y 690.275,Z 783.31,A -85,B 0,C 180,E1 3918.825,E2 3918.825} C_VEL
LIN {X 0,Y 690.342,Z 783.31,A -85,B 0,C 180,E1 3924.297,E2 3924.297} C_VEL
LIN {X 0,Y 690.407,Z 783.31,A -85,B 0,C 180,E1 3929.693,E2 3929.693} C_VEL
LIN {X 0,Y 690.605,Z 783.31,A -85,B 0,C 180,E1 3934.093,E2 3934.093} C_VEL
LIN {X 0,Y 690.576,Z 783.31,A -85,B 0,C 180,E1 3938.107,E2 3938.107} C_VEL
LIN {X 0,Y 690.627,Z 783.31,A -85,B 0,C 180,E1 3943.435,E2 3943.435} C_VEL
LIN {X 0,Y 690.668,Z 783.31,A -85,B 0,C 180,E1 3948.619,E2 3948.619} C_VEL
LIN {X 0,Y 690.742,Z 783.31,A -85,B 0,C 180,E1 3953.709,E2 3953.709} C_VEL
LIN {X 0,Y 690.675,Z 783.31,A -85,B 0,C 180,E1 3958.748,E2 3958.748} C_VEL
LIN {X 0,Y 690.678,Z 783.31,A -85,B 0,C 180,E1 3962.519,E2 3962.519} C_VEL
LIN {X 0,Y 690.687,Z 783.31,A -85,B 0,C 180,E1 3966.301,E2 3966.301} C_VEL
LIN {X 0,Y 690.637,Z 783.31,A -85,B 0,C 180,E1 3971.391,E2 3971.391} C_VEL
LIN {X 0,Y 690.63,Z 783.31,A -85,B 0,C 180,E1 3976.574,E2 3976.574} C_VEL
LIN {X 0,Y 690.492,Z 783.31,A -85,B 0,C 180,E1 3981.906,E2 3981.906} C_VEL
LIN {X 0,Y 690.471,Z 783.31,A -85,B 0,C 180,E1 3986.035,E2 3986.035} C_VEL
LIN {X 0,Y 690.423,Z 783.31,A -85,B 0,C 180,E1 3991.146,E2 3991.146} C_VEL
LIN {X 0,Y 690.396,Z 783.31,A -85,B 0,C 180,E1 3996.34,E2 3996.34} C_VEL
LIN {X 0,Y 690.321,Z 783.31,A -85,B 0,C 180,E1 4001.735,E2 4001.735} C_VEL
LIN {X 0,Y 690.326,Z 783.31,A -85,B 0,C 180,E1 4006.412,E2 4006.412} C_VEL
LIN {X 0,Y 690.312,Z 783.31,A -85,B 0,C 180,E1 4012.202,E2 4012.202} C_VEL
LIN {X 0,Y 690.345,Z 783.31,A -85,B 0,C 180,E1 4016.724,E2 4016.724} C_VEL
LIN {X 0,Y 690.55,Z 783.31,A -85,B 0,C 180,E1 4020.561,E2 4020.561} C_VEL
LIN {X 0,Y 699.307,Z 805.366,A -85,B 0,C 180,E1 4021.222,E2 4021.222} C_VEL
LIN {X 0,Y 698.967,Z 865.73,A -85,B 0,C 180,E1 4022.03,E2 4022.03} C_VEL
LIN {X 0,Y 697.964,Z 908.596,A -85,B 0,C 180,E1 4023.13,E2 4023.13} C_VEL
LIN {X 0,Y 696.545,Z 950.264,A -85,B 0,C 180,E1 4024.755,E2 4024.755} C_VEL
LIN {X 0,Y 695.049,Z 989.753,A -85,B 0,C 180,E1 4026.898,E2 4026.898} C_VEL
LIN {X 0,Y 693.643,Z 1024.256,A -85,B 0,C 180,E1 4029.378,E2 4029.378} C_VEL
LIN {X 0,Y 692.493,Z 1055.723,A -85,B 0,C 180,E1 4032.328,E2 4032.328} C_VEL
LIN {X 0,Y 691.726,Z 1080.945,A -85,B 0,C 180,E1 4035.411,E2 4035.411} C_VEL
LIN {X 0,Y 691.264,Z 1100.684,A -85,B 0,C 180,E1 4038.624,E2 4038.624} C_VEL
LIN {X 0,Y 691.025,Z 1115.931,A -85,B 0,C 180,E1 4042.125,E2 4042.125} C_VEL
LIN {X 0,Y 690.98,Z 1124.073,A -85,B 0,C 180,E1 4044.969,E2 4044.969} C_VEL
LIN {X 0,Y 691.014,Z 1128.176,A -85,B 0,C 180,E1 4047.488,E2 4047.488} C_VEL
LIN {X 0,Y 691.031,Z 1129.121,A -85,B 0,C 180,E1 4051.257,E2 4051.257} C_VEL
LIN {X 0,Y 690.992,Z 1125.286,A -85,B 0,C 180,E1 4054.313,E2 4054.313} C_VEL
LIN {X 0,Y 691.088,Z 1116.746,A -85,B 0,C 180,E1 4057.56,E2 4057.56} C_VEL
LIN {X 0,Y 691.271,Z 1101.913,A -85,B 0,C 180,E1 4061.058,E2 4061.058} C_VEL
LIN {X 0,Y 691.749,Z 1080.269,A -85,B 0,C 180,E1 4064.59,E2 4064.59} C_VEL
LIN {X 0,Y 692.498,Z 1054.894,A -85,B 0,C 180,E1 4067.674,E2 4067.674} C_VEL
LIN {X 0,Y 693.703,Z 1023.1,A -85,B 0,C 180,E1 4070.623,E2 4070.623} C_VEL
LIN {X 0,Y 695.093,Z 988.265,A -85,B 0,C 180,E1 4073.103,E2 4073.103} C_VEL
LIN {X 0,Y 696.613,Z 949.12,A -85,B 0,C 180,E1 4075.205,E2 4075.205} C_VEL
LIN {X 0,Y 697.934,Z 908.788,A -85,B 0,C 180,E1 4076.775,E2 4076.775} C_VEL
LIN {X 0,Y 698.941,Z 866.185,A -85,B 0,C 180,E1 4077.871,E2 4077.871} C_VEL
LIN {X 0,Y 699.113,Z 804.383,A -85,B 0,C 180,E1 4078.708,E2 4078.708} C_VEL
LIN {X 0,Y 690.582,Z 783.31,A -85,B 0,C 180,E1 4079.372,E2 4079.372} C_VEL
LIN {X 0,Y 690.387,Z 783.31,A -85,B 0,C 180,E1 4084.794,E2 4084.794} C_VEL
LIN {X 0,Y 690.259,Z 783.31,A -85,B 0,C 180,E1 4089.8,E2 4089.8} C_VEL
LIN {X 0,Y 690.44,Z 783.31,A -85,B 0,C 180,E1 4094.608,E2 4094.608} C_VEL
LIN {X 0,Y 690.267,Z 783.31,A -85,B 0,C 180,E1 4100.2,E2 4100.2} C_VEL
LIN {X 0,Y 690.319,Z 783.31,A -85,B 0,C 180,E1 4105.201,E2 4105.201} C_VEL
LIN {X 0,Y 690.395,Z 783.31,A -85,B 0,C 180,E1 4109.682,E2 4109.682} C_VEL
LIN {X 0,Y 690.555,Z 783.31,A -85,B 0,C 180,E1 4114.107,E2 4114.107} C_VEL
LIN {X 0,Y 690.537,Z 783.31,A -85,B 0,C 180,E1 4118.096,E2 4118.096} C_VEL
LIN {X 0,Y 690.633,Z 783.31,A -85,B 0,C 180,E1 4123.426,E2 4123.426} C_VEL
LIN {X 0,Y 690.699,Z 783.31,A -85,B 0,C 180,E1 4128.61,E2 4128.61} C_VEL
LIN {X 0,Y 690.793,Z 783.31,A -85,B 0,C 180,E1 4133.7,E2 4133.7} C_VEL
LIN {X 0,Y 690.71,Z 783.31,A -85,B 0,C 180,E1 4138.738,E2 4138.738} C_VEL
LIN {X 0,Y 690.681,Z 783.31,A -85,B 0,C 180,E1 4142.51,E2 4142.51} C_VEL
LIN {X 0,Y 690.665,Z 783.31,A -85,B 0,C 180,E1 4146.292,E2 4146.292} C_VEL
